	xSetForceError:BOOL;
	diSetForceErrorNr:DINT;
	xUpdateErrorList: BOOL;
	xResetErrorWarning:BOOL;
	xHideObject:BOOL;	(* Dies muss aktiv gesetzt werden sobald ein Overlay Message Aktiv ist, ansonsten kann es Probleme geben mit der Annahme der Button *)
(* Sicherheitstüre Maschine und Lader *)
	xOpenSecurityDoorMachine:BOOL;				(* Aufforderung für das Öffnen der Sicherheitstüren *)
	xCloseSecurityDoorMachine:BOOL;				(* Aufforderung für das Schliessen der Sicherheitstüren *)
(* Sicherheitssignale *)
	iSetupMode:INT;								(* Einrichtbetriebswahlschalter
													1=Einrichtbetrieb A
													2=Einrichtbetrieb B
												*)
	xSetupOperateModeActive:BOOL;				(* FALSE=NormalBetrieb, TRUE=Einrichtbetrieb *)
	bStateSafetyCtrl:BYTE;							(*
													0=< Keine Meldung >
													1=< Maschine ist am aufstarten... >
													2=< FreigabeTaste drücken >
													3=< StartTaste drücken >
													4=< Maschinen- und LadeTüre schliessen >
													5=< MaschinenTüren schliessen >
													6=< LadeTüre schliessen >
													7=< Für Positionsfahrt StartTaste drücken   >
													8=< Für Drehbewegung StartTaste drücken  >
													9=< Funktion in Ausführung >
													10=< Funktion in Ausführung...MMI ist blockiert >
													11=< Achsenposition wird überprüft...MMI ist blockiert >
													12=< Servo für Z Achsen stehen nicht bereit >
													13=< Servo für T Achse steht nicht bereit >
													14=< Servo für X Achse steht nicht bereit >
													15=< Kühlmittelpumpe Überlastschutz aktiv >
													16=< Kühlmittelpumpe nicht angeschlossen >
													17=< AntriebSperrTaste deaktivieren >
													18=< Schlüsselschalter deaktivieren >
													19=< Not Aus Taster deaktivieren >
													20=< Zustimmschalter deaktivieren >
													21=< Zustimmschalter aktivieren oder Türen schliessen >
													22=< Zylinderbewegung EIN/AUS drücken >
													23=< Ventile EIN/AUS drücken >
													24=< Zustimmschalter anschliessen >
													25=< Automat in Ausführung >
													26=< Masch.Ref/Grundstellung in Ausführung >
													27=< WstkEntladen in Ausführung >
													28=< HandBetrieb in Ausführung >
													29=< MaschinenTüreOben schliessen >
													30=< MaschinenTüreUnten schliessen >
													31=< MaschinenTüreOben und LadeTüre schliessen >
													32=< MaschinenTüreUnten und LadeTüre schliessen >
												*)
	xHideSafetyCtrlMessage:BOOL;					(* Unterdrückung der Sicherheitsmeldungen "bStateSafetyCtrl" *)
	xNormalOperate_EnergyON:BOOL;
	xSetupOperateA_EnergyON:BOOL;
	xSetupOperateB_EnergyON:BOOL;
	xDeactivateLamp:BOOL;						(* Gilt für den Lampentest, damit der Ausgang nicht mit der Logik überschrieben wird *)
	xSecurityDoorOpen:BOOL;						(* Maschinentüren und/oder Ladetüre offen *)
	bMachineDoorUpState:BYTE;					(* Zustand der Maschinentüre oben 1=Geöffnet, 2=Geschlossen, 3=Fehlverhalten *)
	bMachineDoorChannel1State:BYTE;				(* Zustand des zweikanaligen Türschalter Türe Zu für Türe oben und unten Kanal 1 1=OFF, 2=ON *)
	bMachineDoorChannel2State:BYTE;				(* Zustand des zweikanaligen Türschalter Türe Zu für Türe oben und unten Kanal 2 1=OFF, 2=ON *)
	bMachineDoorUpOpenState:BYTE;				(* Zustand des Türschalter Türe Offen für Türe oben 1=OFF, 2=ON *)
	bMachineDoorInductiveSensorState:BYTE;		(* Zustand des induktiven Sensor für Türe oben 1=OFF, 2=ON *)
	bMachineDoorGuardControlState:BYTE;			(* Zustand der Tür oben Zuhaltung 1=OFF, 2=ON *)
	iMsgInfo_ColourState:INT;						(* 0=Grün, 1=Gelb-->Gelb gilt für Prozess beendet mit mindestens einem Loch NoGo *)
END_STRUCT
END_TYPE

(* Data type in VISUALISIERUNG *)
TYPE ST_EXCHG_SPINDLEBURNIN :
STRUCT
	rTimeActive:REAL;
	rTimeInactive:REAL;
	rTimeMaxActiveFunction:REAL;
	rSpeed_Axis_S:REAL;
	tTimeElapsed:TIME;
END_STRUCT
END_TYPE

(* Data type in VISUALISIERUNG *)
TYPE ST_EXCHG_STATION :
STRUCT
	xExist:BOOL;
	xActiv:BOOL;
	wState:WORD;
	iProfile:INT;
	diErrorNr:DINT;
	sProfileName:STRING(30);
	bAutomodeState:BYTE;
END_STRUCT
END_TYPE

(* Data type in VISUALISIERUNG *)
TYPE ST_EXCHG_STATION_COMMON :
STRUCT
(* State *)
	wState:DWORD;

	T_Param_Machine:ST_RETAIN_DATA_MACHINE;
	T_Param_StationWork:ST_RETAIN_DATA_STATIONWORK;	(* Gilt für MicroHead-  Station *)

	T_ToolCounter_St1:ST_EXCHG_PARAM_TOOLCOUNTER;			(* Braucht es wegen der Parameterliste im NormalBetrieb, da auf diese Parameter gleichzeitig zugegriffen werden muss *)
	T_WPCounter_St1:ST_EXCHG_PARAM_WPCOUNTER;				(* Braucht es wegen der Parameterliste im NormalBetrieb, da auf diese Parameter gleichzeitig zugegriffen werden muss *)

(* Page Quality *)
	T_Button_Quality_Backward:ST_EXCHG_TOUCHBUTTON;
	T_Button_Quality_Forward:ST_EXCHG_TOUCHBUTTON;
	T_Input_Quality_HoleNumber:ST_EXCHG_TOUCHINPUT;

(* Axis State *)
	bState_Axis_Z:BYTE;

(* Gilt für die Ersteinrichtung der Z Achse *)
	iZAxisFirstSetup_StepNr:INT;
	iZAxisFirstSetupStartButton_StepNr:INT;
	iZAxisFirstSetup_ShowObjectNr:INT;
	xInitial_FirstSetupZ:BOOL;		(* TRUE = Ersteinrichtung Z durchgeführt *)
	rZAxisFirstSetup_OffsetSpinToDeskTop:REAL;

	xBlockSelectAutoMode:BOOL;	(* Bei aktivem Prozess muss die Auswahl blockiert sein *)

	(* Disablen von Objekten, wenn es den SystemLevel braucht *)
	xSystemLevelActive:BOOL;

	bActiveStation_St1St2:BYTE;	(* 	0=Arbeitsstation St1St2 Automat nicht Aktiv
									1=Arbeitsstation St1St2 Automat Aktiv
									2=Arbeitsstation St1St2 Automat Fehler *)

(* Gilt für das Aufzeichnen der Rotationsdauer der Spindel *)
	tSpindelActiveRotationTime:TIME;
	iSpindelActiveRotationDay:INT;

	xOnlineValueModified_St1:BOOL;

	xToolSpindle_L_Connect:BOOL;

(* Auswahl der Zylinderkonfiguration *)
	bSelectCylinderConfig:BYTE;		(* 1=Auslenkzylinder, 2=Drehmomentzylinder *)
	bShowCylinderConfig:BYTE;		(* 1=Auslenkzylinder (SM), 2=Auslenkzylinder (L), 3=Drehmomentzylinder (SM), 4=Drehmomentzylinder (L) *)

(* Auswahl der Erst Einrichtung Z Achse *)
	bSelectZAxisProcedure:BYTE;		(* 1=Ersteinrichtung Relation Z-Achse zu oberes Führungsrohr, 2=Ersteinrichtung Z Achse *)
	xBlockSelectZAxisProcedure:BOOL;

(* Gilt für die Ersteinrichtung der Z Achse für die Relation zwischen Z Achse und oberes Führungsrohr *)
	iZAxisGuideTube_StepNr:INT;
	iZAxisGuideTubeStartButton_StepNr:INT;
	iZAxisGuideTube_ShowObjectNr:INT;

(* Bestimmung der Schwingungsqualität der Wippe der Drehmomentüberwachung *)
	rRockerQuality:REAL;
	rRockerQualityMin:REAL;
	rRockerQualityMax:REAL;
	rRockerAmplitude:REAL;
	rRockerAmplitudeMin:REAL;
	rRockerAmplitudeMax:REAL;
	rRockerPosition:REAL;
	diRockerCountHC:DINT;
	diRockerCountHCTime:DINT;

(* Konfiguration der Positionen *)
	iSelectConfigPosition:INT;
	xDisableConfigPosition:BOOL;


(* Regler *)
	rSpeedZ_V1:REAL;					(* IGS *)
	rSpeedZ_V3:REAL;					(* IGS *)
	rTorqueZ_S1:REAL;					(* IGS *)
	rTorqueZ_S4:REAL;					(* IGS *)

	iProgressBar_Torque:INT;				(* IGS *)
	iProgressBar_ZPos:INT;				(* IGS *)
	iProgressBar_ZVel:INT;				(* IGS *)

	xTorqueAfterHC_Min_Overlimit:BOOL;	(* IGS *)
	xTorqueAfterHC_Max_Overlimit: BOOL;	(* IGS *)

	rActual_Torque:REAL;			(* Aktuelles Drehmoment der Drehmomentfeder in mNm - Wechselkopf unabhängig *)	(* IGS *)
	rMaxTorque:REAL;					(* IGS *)

(* Zentrieren *)
	diCentringNumberHCinWindow:DINT;	(* Anzeigen des Zählerstandes wie oft HC in einem definierten Fenster schon eingetroffen ist *)
	xShowSelectCentringProcess:BOOL;	(* Auswahl des Zentrierprozess nur dann zeigen wenn effektiv der Zentrierprozess angewählt ist *)

	rPositionEndProcCalc:REAL;	(* Anzeige oder Eingabe für berechnete EndPosition *)
	xDisableChangeEndPos:BOOL;

	rCentringEndProcCalc:REAL;	(* Anzeige oder Eingabe für berechnete EndPosition *)
	xDisableCentringChangeEndPos:BOOL;

	bSelectShowIncValue:BYTE;	(* 0=Anzeigen der Bearb Ink Werte, 1=Anzeigen der Zentrier Ink Werte *)

	rController2_MinSpeed:REAL;

	rZPositionEndProc:REAL;

	xProcessCylindricalAreaActive:BOOL;

	xSControllerActive:BOOL;
	xOControllerActive:BOOL;
END_STRUCT
END_TYPE

(* Data type in VISUALISIERUNG *)
TYPE ST_EXCHG_TOUCHBUTTON :
STRUCT
	xActive:BOOL;
	xDisable:BOOL;
	xHide:BOOL;
	bState:BYTE;
END_STRUCT
END_TYPE

(* Data type in VISUALISIERUNG *)
TYPE ST_EXCHG_TOUCHINPUT :
STRUCT
	diInput1:DINT;
	diInput2:DINT;
	diInputMin:DINT;
	diInputMax:DINT;
	xDisable:BOOL;
	xChangeColour:BOOL;
END_STRUCT
END_TYPE

(* Data type in VISUALISIERUNG *)
TYPE ST_EXCHG_TOUCHSCREENBTPANEL :
STRUCT
	iNotMaskTextBt:INT;
	iActivBtLeft:INT;
	iStateBtLeft:INT;
	iActivBtRight:INT;
	iStateSetupLamp:INT;
	iStateButtonPage:INT;
	iSelectStationNumber:INT;
END_STRUCT
END_TYPE

(* Data type in VISUALISIERUNG *)
TYPE ST_EXCHG_TOUCHSCREENNAVPANEL :
STRUCT
	wState:WORD;
	wNotMasktext:WORD;
	wActivBt:WORD;
END_STRUCT
END_TYPE

(* Data type in VISUALISIERUNG *)
TYPE ST_EXCHG_VISU :
STRUCT
(* Message structure *)
	T_Message:ST_EXCHG_MESSAGE;
(* Error List Structure *)
	T_MsgErrorEnglish:ST_EXCHG_MESSAGE_LIST;
	T_MsgErrorDeutsch:ST_EXCHG_MESSAGE_LIST;
(* Level structure *)
	T_Level:ST_EXCHG_LEVEL;
(* Variable *)
	iQVisActivNewPage:INT:=0;
	iLoadingStartPage:INT:=1;
	iHeaderTitlePageNumber:INT;
	bActivStation:BYTE:=0;
	bActiveSetupMode:BYTE:=0;	(* 0=AutoMode, 1=SetupMode A, 2=SetupMode B, 3=SetupMode C *)
	bMachineState:BYTE;	(* 1=Ready, no movement, 2=busy function,process or actuator active, 4=Error *)
	xKey_Enter:BOOL;
	xKey_Escape:BOOL;
	xLoadingProcessDone:BOOL;
	sSWVersion:STRING(10):='V4620699';		(* V4620699.pro *)
	sQVisVersion:STRING(10):='V462069902';	(* V4620699_02.qpr-->wird per NovRAM definiert *)
	sHWVersion:STRING(10):='V462069902';		(* V4620699_02.tsm *)
	sIPAddress:STRING(23):='xxx.xxx.xxx.xxx.xxx.xxx';
	sSubNetMask:STRING(23):='xxx.xxx.xxx.xxx.xxx.xxx';
	sGatewayAddress:STRING(23):='xxx.xxx.xxx.xxx.xxx.xxx';
	sAmsNetID:STRING(23):='xxx.xxx.xxx.xxx.xxx.xxx';
	sHostName:STRING(23):='xxxxxxxxxxxxxxxxxxxxxxx';
	xDHCPActive:BOOL:=FALSE;
	xNoRemoteControlActive:BOOL;	(* TRUE = Kein Rechner an der CX2020 angeschlossen *)
	xActiveProcessState_St1St2:BOOL;	(* Ausgabe ob Prozesszustand Aktiv ist oder nicht *)
END_STRUCT
END_TYPE

(* Data type in VISUALISIERUNG *)
TYPE ST_PAGE :
STRUCT
	iIndexConfigPage:INT:=0;
END_STRUCT
END_TYPE

(* Data type in VISUALISIERUNG *)
TYPE ST_QVIS :
STRUCT
	T_PageIndex:ARRAY[0..999] OF ST_PAGE;
	T_ConfigPage:ARRAY[1..csiMaxPage] OF ST_CONFIGPAGE;
	T_CtrleVisu:ST_CTRLEVISU;
	T_PlcParam:ST_VISU_PLC_PARAM;
	T_CtrleAction:ST_CTRLEACTION;
	T_CtrleProcess:ST_CTRLEPROCESS;
END_STRUCT
END_TYPE

(* Data type in VISUALISIERUNG *)
TYPE ST_QVIS_EXCHG_PARAM :
STRUCT
	byOverride:BYTE;					(*Maschinengeschwindigkeit*)
	T_Visu:ST_EXCHG_VISU;
	T_TouchScreenBtPanel:ST_EXCHG_TOUCHSCREENBTPANEL;
	T_BtFunctionPanel:ST_EXCHG_BTFUNCTIONPANEL;
	T_BtParameterList:ST_EXCHG_BTPARAMETERLIST;
	T_TouchScreenNavPanel:ST_EXCHG_TOUCHSCREENNAVPANEL;
	T_Config:ST_EXCHG_CONFIG;
	T_TeachIn:ST_EXCHG_AXIS;
	T_Cylinder:ST_EXCHG_CYLINDER;
	T_Station1:ST_EXCHG_STATION;	(* BearbStation St1 *)
	T_StationCommon:ST_EXCHG_STATION_COMMON;
	T_FunctionCommon:ST_EXCHG_FUNCTION_COMMON;
	T_AnalogSensTorque:ST_EXCHG_ANALOGSENSOR;
	T_ProfileCommon:ST_EXCHG_PROFILE_COMMON;
	T_PartQuality:ST_EXCHG_PARTQUALITY;
	T_LampTest:ST_EXCHG_LAMPTEST;
	T_SpindleBurnIn:ST_EXCHG_SPINDLEBURNIN;
	T_SafetyCtrl:ST_EXCHG_SAFETY_CTRL;
	T_ParamBIOS:ST_EXCHG_PARAM_BIOS;
	xShutdownSystem:BOOL;
	xBIOSButton:BOOL;
	xBIOSButtonHide:BOOL;

	(* Spindelkopf Auswahl Beckhoff/Maxon *)
	xInputSelectAxisSuccesful:BOOL;								(* IGS *)
	xButtonSelect_S1:BOOL;			(* Maxon Spindel *)			(* IGS *)
	xButtonSelect_S2:BOOL;			(* Beckhoff Spindel L *)			(* IGS *)
	xButtonSelect_S3:BOOL;			(* Beckhoff Spindel M *)			(* IGS *)
	xButtonDisable:BOOL;											(* IGS *)
	xWriteSoEParameter:BOOL;									(* IGS *)
	bToolSpindleActive:BYTE;			(*	1 = Maxon Spindel
										2 = Beckhoff Spindel L
										3 = Beckhoff Spindel M *)
END_STRUCT
END_TYPE

(* Data type in VISUALISIERUNG *)
TYPE ST_QVISCTRLE :
STRUCT
	dwInCommand:DWORD;
	dwInCount:DWORD;
	dwInQVisCtrlAddress:DWORD;
	dwInParameterAddress:DWORD;
	dwOutCount:DWORD;
	diOutStatus:DINT;
END_STRUCT
END_TYPE

(* Data type in VISUALISIERUNG *)
TYPE ST_TEMP_ACTIVE_STATE :
STRUCT
	iActCyl_SetupB1_St1:INT;		(* Cyl 1, Cyl 2, Cyl 3 *)

	iActValve_SetupB1_St1:INT;		(* Valve 4, Valve 5 *)

	iActCylinderSetup_SetupB1:INT;

	iActAxis_SetupB1_St1:INT;		(* Z, S und O Achse *)

	iActiveProfile:INT;
	iPtrListProfile:INT;
END_STRUCT
END_TYPE

(* Data type in VISUALISIERUNG *)
TYPE ST_VISU_PLC_PARAM :
STRUCT
	dwSetNewPage:DWORD;
	dwActualPage:DWORD;
	dwPreviousPage:DWORD;
END_STRUCT
END_TYPE

(* Data type in VISUALISIERUNG *)
TYPE ST_VISUPAGENUMBER :
STRUCT
(* Start Page *)
	iStart_Page1:INT:=0;
(* BIOS Page *)
	iBIOS_Page1:INT:=1;
	iBIOS_Page2:INT:=2;
(* NormalOperating-->Task 1 *)
	iAutoMode_Process:INT:=10;
	iAutoMode_ProcessValue1:INT:=11;		(* IGS *)
	iAutoMode_ProcessValue2:INT:=12;		(* IGS *)
	iAutoMode_PartQuality:INT:=13;			(* alt 12 *)
(* NormalOperating-->Task 2 *)
	iAutoMode_Referencing:INT:=20;
(* NormalOperating-->Task3 *)
	iAutoMode_Profile:INT:=30;
(* NormalOperating-->Task 4 *)
	iAutoMode_ToolChange:INT:=40;
	iAutoMode_UserLevel:INT:=41;
	iAutoMode_Language:INT:=42;
(* NormalOperating-->Task 5 *)
	iAutoMode_WPCounter:INT:=50;
	iAutoMode_LampTest:INT:=51;
	iAutoMode_SafetyCheck:INT:=52;
	iAutoMode_SysInfo:INT:=53;
(* NormalOperating-->Task 6 *)
	iAutoMode_ErrorList:INT:=60;
(* NormalOperating-->Parameter *)
	iAutoMode_Parameter:INT:=70;
(* SetupOperate A-->Task 1 *)
	iHandMode_Process:INT:=110;
	iHandMode_WorkParameter:INT:=111;	(* IGS *)
	iHandMode_RegulatorPara:INT:=112;	(* IGS *)
	iHandMode_OnlineChange:INT:=113;		(* alt 111 *)
	iHandMode_ConfigPosition:INT:=114;		(* alt 112 *)
(* SetupOperate A-->Task 3 *)
	iHandMode_ProfileMngmt1:INT:=120;
(* SetupOperate A-->Task 5 *)
	iHandMode_Setup1:INT:=150;
(* SetupOperate A-->Task 6 *)
	iHandMode_ErrorList:INT:=160;
(* SetupOperate A-->Parameter *)
	iHandMode_Parameter:INT:=170;
(* SetupOperate B-->Task 1 *)
	iWorkStation_Axis1:INT:=210;
(* SetupOperate B-->Task 2 *)
	iWorkStation_Cylinder1:INT:=220;
(* SetupOperate B-->Task 3 *)
	iWorkStation_Valve1:INT:=230;
(* SetupOperate B-->Task 4 *)
	iWorkStation_Function1:INT:=240;
(* SetupOperate B-->Task 5 *)
	iWorkStation_Setup1:INT:=250;
	iWorkStation_Setup2:INT:=251;
	iWorkStation_Setup3:INT:=252;
	iWorkStation_Setup4:INT:=253;
	iWorkStation_Setup5:INT:=254;
(* SetupOperate B-->Task 6 *)
	iWorkStation_ErrorList:INT:=260;
(* SetupOperate B-->Parameter *)
	iWorkStation_Parameter:INT:=270;
(* WaitCom_Page1 *)
	iWaitCom_Page1:INT:=1001;
END_STRUCT
END_TYPE

(* POU PRG_STARTUP, ST *)
PROGRAM PRG_STARTUP
VAR
	xPLCWait: BOOL := TRUE;
	TONPLCWait: TON;
	FBInitErrorList:FB_InitErrorList;
	RisingEdgeExecute:R_TRIG;
	iStepFunction: INT;
	xInitVisu: BOOL;
	tTimeOutFunction: TIME;
	xLoading: BOOL;
	TONStartUp: TON;
	xEmergency: BOOL;
	xStartBooting: BOOL;
	xNoAirPressure: BOOL;
	xReadHardware: BOOL;
	xActiveErrorMsg: BOOL;
	iMsgNumber: INT;
	xActiveInfoMsg: BOOL;
	TimerFunction: TON;
	xNovRamParameterReaded: BOOL;
	xTmp: BOOL;
	TONWaitResetOutput: TON;
	RisingEdgeStartButton: R_TRIG;
	RisingEdgeQuitButton: R_TRIG;
	xDeleteErrorMessage: BOOL;
	TONWaitCircuitOn: TON;
	xMsgActiveDeactivatedSupply: BOOL;
	xStationErrorActive: BOOL;
	tTimeStartUp: TIME := T#40ms;
	xActiveBootingError: BOOL;
	xForceCloseMessage: BOOL;
	xActiveWarningMsg: BOOL;
	xSetOutputDisable: BOOL;
	iStepFunctionMsg: INT;
	xActiveInfoMsgIntern: BOOL;
	xActiveErrorMsgIntern: BOOL;
	xActiveWarningMsgIntern: BOOL;
	TONWaitMessage: TON;
	iStepFunctionON: INT;
	TONWaitSetSecStateON: TON;
	xSwitchOffStartUpFunction: BOOL;
	xMachineActivated: BOOL;
	iStepUPS: INT;
	xFallingEdgeEnergyOff:BOOL;
	xRisingEdgeEnergyOn:BOOL;
	TONWaitEndMessage: TON;
	RisingEdgePower_SetupA_St1: R_TRIG;
	FallingEdgePower_SetupA_St1: F_TRIG;
	RisingEdgePower_SetupB_St1: R_TRIG;
	FallingEdgePower_SetupB_St1: F_TRIG;
	FBSafetyLogic: FB_SAFETYLOGIC;
	ptrTCommonAxis : POINTER TO ST_AXIS;
	xInitPointer: BOOL;
	FBCheckMachineState: FB_CHECKMACHINESTATE;
	iStepCheckSafetyError: INT;
	xTwinSAFEError: BOOL;
	xCheckConfirm: BOOL;
	xTerminalError: BOOL;
	RisingEdgePower_NormalOperate_St1St2: R_TRIG;
	FallingEdgePower_NormalOperate_St1St2: F_TRIG;
	FBGetAdaptersInfo: FB_GetAdaptersInfo;
	ii: INT;
	xReadyToCheckSafety: BOOL;
	xFirstBooting: BOOL;
	fbNT_Shutdown: NT_Shutdown;
	FBBIOSPARAMETER: FB_BIOSPARAMETER;
	xNovRamError: BOOL;
	RisingEdgeOpenSecDoorMachine: R_TRIG;
	RisingEdgeCloseSecDoorMachine: R_TRIG;
	xOpenSecurityDoor: BOOL;
	xCloseSecurityDoor: BOOL;
	iStepOpenSecurityDoor: INT;
	TONWaitSecurityDoorLocked: TON;
	iStepCloseSecurityDoor: INT;
	xReadySetMessageDeactivate: BOOL;
	xReadySetMessageActivate: BOOL;
	TONWaitCheckAirPressure: TON;
	RisingEdgeUPS: R_TRIG;
	TONPrellen_ON: TON;
	TONPrellen_OFF: TON;
	xCabinDoorLocked: BOOL;
	xInitMachineLamp: BOOL;
	RisingEdgeFirstTime: R_TRIG;
	RisingEdgeSetupOperateMode: R_TRIG;
	xInit: BOOL;
	TPEnablingSwitch: TP;
	RisingEdgeCheckSwitchVibration: R_TRIG;
	TONWaitStopVibration: TON;
	wWCEPOS_State: WORD;
	wEtherCAT_2_State: WORD;
	xActivateEPOSPreOPMode: BOOL;
	FBGetHostName: FB_GetHostName;
	FBGetLocalAmsNetId: FB_GetLocalAmsNetId;
	sCopyString: STRING;
	iPoint: INT;
	sCopyStringIP: STRING;

	T_TwinSafeInWithoutHW:POINTER TO	ST_TWINSAFE_IN;
	T_TwinSafeOutWithoutHW:	POINTER TO ST_TWINSAFE_OUT;

	(* .StartUpFunction_Booting *)
	TONWaitMessage1: TON;		(* IGS *)
END_VAR
(****************************************************************************************************************************************************)
(**********      This Functionblock manage the booting of the machine and the security mangament of the machine during   ********)
(**********       the machine operating                           														    ************)
(****************************************************************************************************************************************************)
(* waiting 5 sec before starting *)
	IF xPLCWait THEN
		TONPLCWait(IN:=TRUE,PT:=T#5s);
		IF TONPLCWait.Q THEN
			TONPLCWait(IN:=FALSE);
			xPLCWait:=FALSE;
			T_StartUp.T_Ctrle.xExecute:=FALSE;
			T_StartUp.T_Ctrle.xDone:=FALSE;
			T_StartUp.T_Ctrle.xErr:=FALSE;
			T_StartUp.T_Ctrle.xReset:=FALSE;
			T_StartUp.T_State.xPLCReady:=FALSE;
			T_StartUp.T_Ctrle.iFunction:=0;
			T_StartUp.T_Ctrle.udiErrorID:=16#0;
			T_StartUp.T_State.xBlockChangeMovementVisu:=TRUE;
			T_StartUp.T_Ctrle.iMsgNumber:=0;
			(* activ function "Start PLC" *)
			T_StartUp.T_Ctrle.xExecute:=TRUE;
			T_StartUp.T_Ctrle.iFunction:=1;
			FBInitErrorList(T_ErrorList:= T_ErrorList);	(* Init Static Text for Error List *)
		END_IF;
		RETURN;
	END_IF;
	(* Start and Quit Button *)
	RisingEdgeStartButton(CLK:=IxStartButton);
	RisingEdgeQuitButton(CLK:=IxReleaseButton);
	(* IN<-->OUT --> für TwinSAFE Verbindung mit Standard IO zu Sicherheit IO *)
	TPEnablingSwitch(IN:=	T_TwinSafeIn.IxEnablingSwitchActiveCh1 AND T_TwinSafeIn.IxEnablingSwitchActiveCh2 AND
							(NOT(FBSafetyLogic.xMachineDoorClose)) AND T_StartUp.T_State.xCompleted, PT:=T#0.1s);
	QxTwinSafeReleaseButton:=(IxReleaseButton OR TPEnablingSwitch.Q) ;	(* Übergabe des IxReleaseButton an TwinSafe Logik *)
	CtrlPowerSupply;
	CtrlEmergency;
	CtrlSecurityDoor;
	CtrlSecurityState;
	CtrlBIOSParameter;
	CtrlMachineLamp;
	CtrlStartUpFunction;

	IF NOT(xEmergency) AND NOT(xNoAirPressure) AND NOT(xTerminalError) THEN
		StartUpFunction_Initialisation;
		StartUpFunction_ReadHW;
		StartUpFunction_Booting;
		StartUpFunction_Loading;
	END_IF;

	StartUpFunction_MessageActivate;
	StartUpFunction_Emergency;

(* Delete of the line error message *)
	IF xDeleteErrorMessage THEN
		xDeleteErrorMessage:=FALSE;
		T_ExchgParam.T_Visu.T_Message.sDynamicTextEnglish:='';
		T_ExchgParam.T_Visu.T_Message.sDynamicTextDeutsch:='';
		T_ExchgParam.T_Visu.T_Message.sDynamicTextFrancais:='';
		T_ExchgParam.T_Visu.T_Message.iState:=0;	(* Meldung löschen *)
	END_IF;

(* Set Output disabled *)
	IF xSetOutputDisable THEN
		T_TwinSafeCtrleOUT.xTwinSAFE_Run_1:=FALSE;	(* Stop TwinSafe Groupe *)
		TProcess.T_Ctrle.xEnable:=FALSE;
		QxCtrlLampStartButton:=FALSE;
		QxCtrlLampStopButton:=FALSE;
		QxCtrlLampReleaseButton:=FALSE;
		QxCtrlLampAxesCurrentOff:=FALSE;
		QxReadyToOperateMasterModul1:=FALSE;
		QxReadyToOperateMasterModul2:=FALSE;
		TStation_Work_St1.TControl.xEnable:=FALSE;
		T_ExchgParam.T_Visu.iLoadingStartPage:=1;
		(* confirm *)
		xSetOutputDisable:=FALSE;
	END_IF;

	IF NOT(gxBlockChangeMovementVisuActiveMessage) AND NOT(xEmergency) AND NOT(xNoAirPressure) AND NOT(xTerminalError) AND NOT(xActiveInfoMsg) AND NOT(xActiveInfoMsgIntern)
	AND NOT(xActiveErrorMsg) AND NOT(xActiveErrorMsgIntern) AND NOT(xActiveWarningMsg) AND NOT(xActiveWarningMsgIntern) AND NOT(xPLCWait) AND T_StartUp.T_State.xCompleted THEN
		T_StartUp.T_State.xBlockChangeMovementVisu:=FALSE;
	END_IF;

	IF gxHardwareOFF AND NOT(xInit) THEN
		xInit:=TRUE;

		T_TwinSafeInWithoutHW:=ADR(T_TwinSafeIn);
		T_TwinSafeOutWithoutHW:=ADR(T_TwinSafeOut);
		T_TwinSafeInWithoutHW^.IxAxesCurrentOffCh1:=TRUE;
		T_TwinSafeInWithoutHW^.IxAxesCurrentOffCh2:=TRUE;
		T_TwinSafeInWithoutHW^.IxCabinDoorClose:=TRUE;
		T_TwinSafeInWithoutHW^.IxCabinDoorCloseCh1:=TRUE;
		T_TwinSafeInWithoutHW^.IxCabinDoorCloseCh2:=TRUE;
		T_TwinSafeInWithoutHW^.IxEmergencyStopButtonCh1:=TRUE;
		T_TwinSafeInWithoutHW^.IxEmergencyStopButtonCh2:=TRUE;
		T_TwinSafeInWithoutHW^.IxReadyToOperateMasterModul1:=TRUE;
		T_TwinSafeInWithoutHW^.IxReadyToOperateMasterModul2:=TRUE;
		T_TwinSafeOutWithoutHW^.QxContactor24VCh1:=TRUE;
		T_TwinSafeOutWithoutHW^.QxContactor24VCh2:=TRUE;
		T_TwinSafeOutWithoutHW^.QxContactorMasterModul400VCh1:=TRUE;
		T_TwinSafeOutWithoutHW^.QxContactorMasterModul400VCh2:=TRUE;
		T_TwinSafeOutWithoutHW^.QxEnablingAxisSpindle_St1:=TRUE;
		T_TwinSafeOutWithoutHW^.QxEnablingSwitchLed:=TRUE;

		T_NovRam.T_Parameter.T_StationWork[gciStationSt1].T_AxisState.xReferencedZAxis:=TRUE;

	END_IF;
END_PROGRAM
ACTION CtrlBIOSParameter:
	IF T_StartUp.T_State.xPLCReady THEN
		xTmp:=	T_TwinSafeOut.QxContactorMasterModul400VCh1 AND T_TwinSafeOut.QxContactorMasterModul400VCh2 AND
				T_TwinSafeOut.QxContactor24VCh1;
		FBBIOSPARAMETER(	dwBIOSPasswordPage:= gT_PageNumber.iBIOS_Page1,
							dwBIOSParameterPage:= gT_PageNumber.iBIOS_Page2,
							xActiveCurrentAxes:=xTmp,
							xReadyToSwitchPasswordPage:=xStartBooting AND (iStepFunction <= 40) AND T_TwinSafeIn.IxEmergencyStopButtonCh1 AND T_TwinSafeIn.IxEmergencyStopButtonCh2,
							T_Visu:= T_VisuQVis,
							T_ExchgParam:=T_ExchgParam,
							T_HDD:= T_HDD,
							T_NovRam:= T_NovRam,
							T_CtrlePanel:= T_CtrlePanel);
	END_IF;
END_ACTION
ACTION CtrlEmergency:
(* check the emergency stop, the air pressure, Lightbus of the MasterAxis after booting the machine *)

	IF T_StartUp.T_State.xPLCReady AND NOT(gxHardwareOFF) THEN
	(* check emergency stop, only if it is not already in this state *)
		IF NOT(T_TwinSafeIn.IxEmergencyStopButtonCh1) OR NOT(T_TwinSafeIn.IxEmergencyStopButtonCh2) THEN
			RisingEdgeExecute(CLK:=FALSE);
			(* Set emergency function *)
			T_StartUp.T_Ctrle.xExecute:=TRUE;
			T_StartUp.T_Ctrle.iFunction:=4;
			xSwitchOffStartUpFunction:=TRUE;
		END_IF;

	(* check air pressure, only if it is not already in this state *)
		IF NOT(IxAirSupply) AND T_TwinSafeOut.QxContactor24VCh1 AND T_TwinSafeOut.QxContactor24VCh2 THEN
			TONWaitCheckAirPressure(IN:=T_TwinSafeOut.QxContactor24VCh1 AND T_TwinSafeOut.QxContactor24VCh2,PT:=T#2s);
			IF TONWaitCheckAirPressure.Q THEN
				TONWaitCheckAirPressure(IN:=FALSE);
				(* Set No Air pressure function *)
				T_StartUp.T_Ctrle.xExecute:=TRUE;
				T_StartUp.T_Ctrle.iFunction:=6;
				xSwitchOffStartUpFunction:=TRUE;
			END_IF;
		ELSE
			TONWaitCheckAirPressure(IN:=FALSE);
		END_IF;

		IF xActivateEPOSPreOPMode THEN
			wWCEPOS_State:=8;
			wEtherCAT_2_State:=0;
		ELSE
			wWCEPOS_State:=T_TerminalState.wWCEPOS_State;
			wEtherCAT_2_State:=T_TerminalState.wEtherCAT_2_State;
		END_IF;
	(* Beckhoff Klemmen oder Koppler Überprüfung oder Power Supply 24V *)
		IF NOT(gxHardwareOFF) THEN
			xTmp:=	(T_TerminalState.wEtherCAT_1_State <> 0) OR (wEtherCAT_2_State <> 0) OR (T_TerminalState.wWCMasterAxisModul1_State <> 8) OR (T_TerminalState.wWCMasterAxisModul2_State <> 8)
					OR (wWCEPOS_State <> 8) OR (T_TerminalState.wWCSMCValve <> 8) OR NOT(IxFuse24VDC_OK);
		ELSE
			xTmp:=	FALSE;
		END_IF;
		IF xTmp THEN
			(* Set Terminal Error *)
			T_StartUp.T_Ctrle.xExecute:=TRUE;
			T_StartUp.T_Ctrle.iFunction:=3;
			xSwitchOffStartUpFunction:=TRUE;
		END_IF;

	(* Disable the active StartUp Function *)
		IF xSwitchOffStartUpFunction THEN
			xSwitchOffStartUpFunction:=FALSE;
			xInitVisu:=FALSE;
			xLoading:=FALSE;
			xStartBooting:=FALSE;
			xActiveErrorMsg:=FALSE;
			xActiveInfoMsg:=FALSE;
			xActiveWarningMsg:=FALSE;
			xNoAirPressure:=FALSE;
			xReadHardware:=FALSE;
			xTerminalError:=FALSE;
			T_StartUp.T_State.xCompleted:=FALSE;
		END_IF;
	END_IF;
END_ACTION
ACTION CtrlMachineLamp:
IF NOT(xInitMachineLamp) THEN
	xInitMachineLamp:=TRUE;
	TMachineLamp.T_CtrleCyl.xFBActiv:=TRUE;
	TMachineLamp.T_Config.xActivState:=TRUE;
	TMachineLamp.T_CtrleCyl.xReset:=TRUE;
END_IF;
RisingEdgeFirstTime(CLK:=T_StartUp.T_State.xPLCReady);
IF RisingEdgeFirstTime.Q OR RisingEdgeSetupOperateMode.Q THEN
	(* Einschalten der Einrichtlampe, nachdem die Maschine eingeschaltet wurde *)
	TMachineLamp.T_CtrleCyl.iFunction:=2;
	TMachineLamp.T_CtrleCyl.xExecute:=TRUE;
END_IF;
IF NOT(T_StartUp.T_State.xCompleted) AND T_StartUp.T_State.xPLCReady THEN
	(* Sollte z.B. wegen dem Not Aus die StartSeite wieder erreicht werden, dann muss die Lampe falls sie ausgeschaltet ist wieder eingeschaltet werden *)
	IF NOT(TMachineLamp.T_CtrleCyl.T_Standard.xActivOn) AND NOT(TMachineLamp.T_CtrleCyl.xExecute) AND TMachineLamp.T_CtrleCyl.xDone THEN
		TMachineLamp.T_CtrleCyl.iFunction:=2;
		TMachineLamp.T_CtrleCyl.xExecute:=TRUE;
	END_IF;
END_IF;
END_ACTION
ACTION CtrlPowerSupply:
RisingEdgeUPS(CLK:=TStatusUPS.ePowerStatus = PowerOnBattery);
IF RisingEdgeUPS.Q OR T_ExchgParam.xShutdownSystem THEN
	CASE iStepUPS OF
	1:	T_CtrleUPS.xBlockSystem_PowerFail:=TRUE;	(* Schicht 5 wird gesperrt *)
		T_TwinSafeCtrleOUT.xTwinSAFE_Run_1:=FALSE;	(* Stop TwinSafe Groupe 1 *)
		TProcess.T_Ctrle.xEnable:=FALSE;
		TStation_Work_St1.TControl.xEnable:=FALSE;
		xSwitchOffStartUpFunction:=FALSE;
		xInitVisu:=FALSE;
		xLoading:=FALSE;
		xStartBooting:=FALSE;
		xActiveErrorMsg:=FALSE;
		xActiveInfoMsg:=FALSE;
		xActiveWarningMsg:=FALSE;
		xNoAirPressure:=FALSE;
		xTerminalError:=FALSE;
		xReadHardware:=FALSE;
		T_StartUp.T_State.xCompleted:=FALSE;
		xActiveErrorMsgIntern:=TRUE;
		iStepFunctionMsg:=1;
		IF RisingEdgeUPS.Q THEN
			iMsgNumber:=51;		(* Stromausfall Detektiert! Daten werden im NovRAM gespeichert!! Steuerung ist blockiert! *)
		ELSIF T_ExchgParam.xShutdownSystem THEN
			iMsgNumber:=47;		(* System wird heruntergefahren! Daten werden im NovRAM gespeichert!! Steuerung ist blockiert! *)
		END_IF;
		IF xMachineActivated THEN
			iStepUPS:=iStepUPS + 1;
		ELSE
			fbNT_Shutdown(	NETID:= '127.0.0.1.1.1',
							DELAY:= 1,
							START:= FALSE,
							TMOUT:= T#10s);
			iStepUPS:=4;
		END_IF;
	(* NovRAM speichern *)
	2:	IF NOT(T_NovRAM.T_Ctrle.xExecute) AND (T_NovRAM.T_Ctrle.xDone OR T_NovRAM.T_Ctrle.xErr) THEN
			T_NovRAM.T_Ctrle.xExecute:=TRUE;
			T_NovRAM.T_Ctrle.iFunction:=2;
			iStepUPS:=iStepUPS + 1;
		END_IF;
	3:	IF NOT(T_NovRAM.T_Ctrle.xExecute) AND (T_NovRAM.T_Ctrle.xDone OR T_NovRAM.T_Ctrle.xErr) THEN
			iStepUPS:=iStepUPS + 1;
			fbNT_Shutdown(	NETID:= '127.0.0.1.1.1',
							DELAY:= 1,
							START:= FALSE,
							TMOUT:= T#10s);
		END_IF;
	4:	IF NOT(T_NovRAM.T_Ctrle.xExecute) AND (T_NovRAM.T_Ctrle.xDone OR T_NovRAM.T_Ctrle.xErr) THEN
			fbNT_Shutdown(	NETID:='127.0.0.1.1.1',
							DELAY:= 1,
							START:= TRUE,
							TMOUT:= T#10s);
			IF NOT(fbNT_Shutdown.BUSY) OR fbNT_Shutdown.ERR OR T_ExchgParam.xShutdownSystem THEN
				iStepUPS:=99;	(* CPU kann nun heruntergefahren werden *)
			END_IF;
		END_IF;
	END_CASE;
ELSE
	iStepUPS:=1;
END_IF;
END_ACTION
ACTION CtrlSecurityDoor:
RisingEdgeOpenSecDoorMachine(CLK:=T_ExchgParam.T_SafetyCtrl.xOpenSecurityDoorMachine);
RisingEdgeCloseSecDoorMachine(CLK:=T_ExchgParam.T_SafetyCtrl.xCloseSecurityDoorMachine);
IF RisingEdgeOpenSecDoorMachine.Q THEN
	xOpenSecurityDoor:=TRUE;
	xCloseSecurityDoor:=FALSE;
	T_ExchgParam.T_SafetyCtrl.xCloseSecurityDoorMachine:=FALSE;
END_IF;
IF RisingEdgeCloseSecDoorMachine.Q THEN
	xOpenSecurityDoor:=FALSE;
	xCloseSecurityDoor:=TRUE;
	T_ExchgParam.T_SafetyCtrl.xOpenSecurityDoorMachine:=FALSE;
END_IF;
TONPrellen_ON(IN:=IxCabinDoorLocked,PT:=T#50ms);
TONPrellen_OFF(IN:=NOT(IxCabinDoorLocked),PT:=T#50ms);
IF TONPrellen_ON.Q THEN
	xCabinDoorLocked:=TRUE;
END_IF;
IF TONPrellen_OFF.Q THEN
	xCabinDoorLocked:=FALSE;
END_IF;
IF xOpenSecurityDoor THEN
	CASE iStepOpenSecurityDoor OF
		1:	IF QxCabinDoorLock THEN
				xReadySetMessageDeactivate:=TRUE;
			END_IF;
			QxCabinDoorLock:=FALSE;
			TONWaitSecurityDoorLocked(IN:=FALSE);
			(* next step *)
			iStepOpenSecurityDoor:=iStepOpenSecurityDoor + 1;
		2:	TONWaitSecurityDoorLocked(IN:=TRUE,PT:=T#2000ms);
			IF TONWaitSecurityDoorLocked.Q OR (xCabinDoorLocked) THEN
				TONWaitSecurityDoorLocked(IN:=FALSE);
				(* next step *)
				iStepOpenSecurityDoor:=iStepOpenSecurityDoor + 1;
			END_IF;
		3:	xOpenSecurityDoor:=FALSE;
			T_ExchgParam.T_SafetyCtrl.xOpenSecurityDoorMachine:=FALSE;
			IF NOT(xCabinDoorLocked) THEN	(* IxCabinDoorUpLocked, Check if CabinDoor of the Machine is no more blocked *)
				T_ExchgParam.T_Visu.T_Message.iState:=287;	(* Kabinen-Türe Zuhaltung fehlerhaft beim öffnen ! *)
				xReadySetMessageDeactivate:=FALSE;
			END_IF;
			IF xReadySetMessageDeactivate THEN
				T_ExchgParam.T_Visu.T_Message.iState:=281;	(* Die Zuhaltung der Sicherheitstüren wurde deaktiviert! *)
			END_IF;
	END_CASE;
ELSE
	xReadySetMessageDeactivate:=FALSE;
	iStepOpenSecurityDoor:=1;
END_IF;
IF xCloseSecurityDoor THEN
	CASE iStepCloseSecurityDoor OF
		1:	IF NOT(QxCabinDoorLock) THEN
				xReadySetMessageActivate:=TRUE;
			END_IF;
			QxCabinDoorLock:=TRUE;
			TONWaitSecurityDoorLocked(IN:=FALSE);
			(* next step *)
			iStepCloseSecurityDoor:=iStepCloseSecurityDoor + 1;
		2:	TONWaitSecurityDoorLocked(IN:=TRUE,PT:=T#2000ms);
			IF TONWaitSecurityDoorLocked.Q OR NOT(xCabinDoorLocked) THEN
				TONWaitSecurityDoorLocked(IN:=FALSE);
				(* next step *)
				iStepCloseSecurityDoor:=iStepCloseSecurityDoor + 1;
			END_IF;
		3:	xCloseSecurityDoor:=FALSE;
			T_ExchgParam.T_SafetyCtrl.xCloseSecurityDoorMachine:=FALSE;
			IF xCabinDoorLocked THEN	(* IxCabinDoorUpLocked, Check if CabinDoor of the Machine is blocked *)
				T_ExchgParam.T_Visu.T_Message.iState:=286;	(* Kabinen-Türe Zuhaltung fehlerhaft beim schliessen ! *)
				xReadySetMessageActivate:=FALSE;
			END_IF;
			IF xReadySetMessageActivate THEN
				T_ExchgParam.T_Visu.T_Message.iState:=280;	(* Die Zuhaltung der Sicherheitstüren wurde aktiviert! *)
			END_IF;
	END_CASE;
ELSE
	xReadySetMessageActivate:=FALSE;
	iStepCloseSecurityDoor:=1;
END_IF;
END_ACTION
ACTION CtrlSecurityState:
	IF NOT(xInitPointer) THEN
		xInitPointer:=TRUE;
		ptrTCommonAxis:=ADR(TStation_Work_St1.THWWorkStation.TAxisZ);
	END_IF;
(* Function for Switch on the Security State *)
	IF T_StartUp.T_Ctrle.xSetSecurityStateON THEN
		CASE iStepFunctionON OF
		1:	QxCtrlLampStartButton:=FALSE;
			QxCtrlLampStopButton:=FALSE;
			QxCtrlLampReleaseButton:=FALSE;
			QxCtrlLampAxesCurrentOff:=FALSE;
			TONWaitSetSecStateON(IN:=FALSE);
			iStepFunctionON:=2;
		2:	TONWaitSetSecStateON(IN:=TRUE,PT:=T#500ms);
			IF TONWaitSetSecStateON.Q THEN
				TONWaitSetSecStateON(IN:=FALSE);
				T_TwinSafeCtrleOUT.xTwinSAFE_Run_1:=FALSE;	(* Stop TwinSafe Groupe 1 *)
				iStepFunctionON:=3;
			END_IF;
		3:	TONWaitSetSecStateON(IN:=TRUE,PT:=T#500ms);
			IF TONWaitSetSecStateON.Q THEN
				TONWaitSetSecStateON(IN:=FALSE);
				iStepFunctionON:=4;
			END_IF;
		4:	T_TwinSafeCtrleOUT.xTwinSAFE_Run_1:=TRUE;	(* Start TwinSafe Groupe 1 *)
			T_StartUp.T_Ctrle.xSetSecurityStateON:=FALSE;
			TONWaitSetSecStateON(IN:=FALSE);
			iStepFunctionON:=1;
		END_CASE;
	ELSE
		iStepFunctionON:=1;
		TONWaitSetSecStateON(IN:=FALSE);
	END_IF;

(* Zustandsüberwachung und Zuordnung der Sicherheitssignale *)
FBSafetyLogic(	T_TwinSafeIn:=T_TwinSafeIn,
				T_TwinSafeOut:=T_TwinSafeOut,
				xActiveBooting:=xLoading,
				xActiveBootingError:=xActiveBootingError,
				xVisuFunctionActive:=(NOT(T_VisuQVis.T_CtrleAction.xDone) OR T_VisuQVis.T_CtrleAction.xFunctionActive),
				dwActualPage:= T_VisuQVis.T_PlcParam.dwActualPage,
				xOverlayMessageAcitve:=(T_ExchgParam.T_SafetyCtrl.bStateMessageError<>0) OR (T_ExchgParam.T_SafetyCtrl.bStateMessageInfo<>0) OR (T_ExchgParam.T_SafetyCtrl.bStateMessageWarning<>0),
				iStateMessage:=T_ExchgParam.T_Visu.T_Message.iState,
				TCommonAxis:=ptrTCommonAxis^);

IF gT_SafetyStatus.xSetupOperateModeActive THEN
	CASE T_ExchgParam.T_TeachIn.iSetup_AxisSel OF
	1:	ptrTCommonAxis:=ADR(TStation_Work_St1.THWWorkStation.TAxisZ);
	2,3:	ptrTCommonAxis:=ADR(TStation_Work_St1.THWWorkStation.TAxisS);
	ELSE
		ptrTCommonAxis:=ADR(TStation_Work_St1.THWWorkStation.TAxisZ);
	END_CASE
END_IF;

IF (T_ExchgParam.T_SafetyCtrl.bStateSafetyCtrl = 99) OR T_ExchgParam.T_Visu.T_Message.xShowMessageInfo OR
    T_ExchgParam.T_Visu.T_Message.xShowMessageInput OR T_ExchgParam.T_Visu.T_Message.xShowMessageWarning OR
    (T_ExchgParam.T_Visu.T_Message.iState = 401) THEN
	T_ExchgParam.T_SafetyCtrl.xHideSafetyCtrlMessage:=TRUE;	(* Sicherheitsstatusmeldung auf der Visualisierung unterdrücken *)
ELSE
	T_ExchgParam.T_SafetyCtrl.xHideSafetyCtrlMessage:=FALSE;
END_IF;

T_ExchgParam.T_SafetyCtrl.bStateSafetyCtrl:=FBSafetyLogic.bStateSafetyCtrl;		(* Ausgabe direkt an der Visualisierung um den Operator Mitteilen zu können, was er unternehmen muss damit er Prozess,Funktion usw. auslösen kann *)

(* Kontrollampe für Freigabe QxCtrlLampReleaseButton der Energieversorgung *)
IF NOT(T_ExchgParam.T_SafetyCtrl.xDeactivateLamp) THEN	(* Wenn Lampen Test Aktiv ist, dann muss dies gesperrt werden *)
	QxCtrlLampReleaseButton:=	NOT(gT_SafetyStatus.xEnergyONNormalMode OR gT_SafetyStatus.xEnergyONSetupModeASt1 OR
								gT_SafetyStatus.xEnergyONSetupModeBSt1) AND
								FBSafetyLogic.xSafetyNotActive AND T_TwinSafeCtrleOUT.xTwinSAFE_Run_1 AND T_StartUp.T_State.xPLCReady AND
								(gT_SafetyStatus.xSecurityDoorClose);
END_IF;

(* Check Power switch on/off from the security circuit for control the Station *)
	RisingEdgePower_NormalOperate_St1St2(CLK:=gT_SafetyStatus.xEnergyONNormalMode);
	FallingEdgePower_NormalOperate_St1St2(CLK:=gT_SafetyStatus.xEnergyONNormalMode);
	RisingEdgePower_SetupA_St1(CLK:=	gT_SafetyStatus.xEnergyONSetupModeASt1);
	FallingEdgePower_SetupA_St1(CLK:=gT_SafetyStatus.xEnergyONSetupModeASt1);
	RisingEdgePower_SetupB_St1(CLK:=gT_SafetyStatus.xEnergyONSetupModeBSt1);
	FallingEdgePower_SetupB_St1(CLK:=gT_SafetyStatus.xEnergyONSetupModeBSt1);

	IF T_StartUp.T_State.xCompleted THEN
		xTmp:=	RisingEdgePower_NormalOperate_St1St2.Q OR FallingEdgePower_NormalOperate_St1St2.Q OR
				RisingEdgePower_SetupA_St1.Q OR FallingEdgePower_SetupA_St1.Q OR
				RisingEdgePower_SetupB_St1.Q OR FallingEdgePower_SetupB_St1.Q;
		IF xTmp THEN
			TStation_Work_St1.TControl.xSecurityCircuitOn:=			RisingEdgePower_NormalOperate_St1St2.Q OR RisingEdgePower_SetupA_St1.Q OR RisingEdgePower_SetupB_St1.Q;
			TStation_Work_St1.TControl.xSecurityCircuitOff:=			FallingEdgePower_NormalOperate_St1St2.Q OR FallingEdgePower_SetupA_St1.Q OR FallingEdgePower_SetupB_St1.Q;
		END_IF;
	(* Message Energy on/off *)
		xRisingEdgeEnergyOn:=	RisingEdgePower_NormalOperate_St1St2.Q OR
								RisingEdgePower_SetupA_St1.Q OR RisingEdgePower_SetupB_St1.Q;

		xFallingEdgeEnergyOff:=	FallingEdgePower_NormalOperate_St1St2.Q OR
								FallingEdgePower_SetupA_St1.Q OR FallingEdgePower_SetupB_St1.Q;

		IF T_StartUp.T_State.xCompleted AND xFallingEdgeEnergyOff THEN
			IF (T_ExchgParam.T_Visu.T_Message.iState = 0) OR (T_ExchgParam.T_Visu.T_Message.iState = 228) THEN
				T_ExchgParam.T_Visu.T_Message.iState:=229;	(* Warnung: Die Energieversorgung ist AUS ! *)
				TONWaitEndMessage(IN:=FALSE);
				T_ExchgParam.T_StationCommon.xBlockSelectAutoMode:=FALSE;
			END_IF;
		END_IF;
		IF T_StartUp.T_State.xCompleted AND xRisingEdgeEnergyOn THEN
			IF (T_ExchgParam.T_Visu.T_Message.iState = 0) OR (T_ExchgParam.T_Visu.T_Message.iState = 229) OR (T_ExchgParam.T_Visu.T_Message.iState = 279) THEN
				T_ExchgParam.T_Visu.T_Message.iState:=228;	(* Warnung: Die Energieversorgung ist EIN ! *)
				TONWaitEndMessage(IN:=FALSE);
			END_IF;
		END_IF;

	END_IF;

(* Überprüfe Maschinenstatus damit die entsprechende LED auf der Visu ausgegeben werden kann *)
FBCheckMachineState(	xSecurityKey:= gT_SafetyStatus.xSetupOperateModeActive,
						iSetupMode:= gT_SafetyStatus.iSetupMode,
						xNormalOperate_EnergyON:= gT_SafetyStatus.xEnergyONNormalMode,
						xSetupOperateA_EnergyON:= gT_SafetyStatus.xEnergyONSetupModeASt1,
						xSetupOperateB_EnergyON:= gT_SafetyStatus.xEnergyONSetupModeBSt1);
T_ExchgParam.T_SafetyCtrl.xNormalOperate_EnergyON:=	gT_SafetyStatus.xEnergyONNormalMode;
T_ExchgParam.T_SafetyCtrl.xSetupOperateA_EnergyON:=	gT_SafetyStatus.xEnergyONSetupModeASt1;
T_ExchgParam.T_SafetyCtrl.xSetupOperateB_EnergyON:=	gT_SafetyStatus.xEnergyONSetupModeBSt1;

(* Überwachung der Not Bremse für alle Achsen die am AX5206 angeschlossen sind beim ausschalten der Energieversorgung *)
	IF IxTwinSafeQuickStopMaster1_1 THEN	(* QuickStop Achsen von TwinSAFE *)
		QxEnableQuickStopMasterModul1:=TRUE;
	ELSE
		QxEnableQuickStopMasterModul1:=FALSE;	(* QxEnableQuickStopMasterModul1-->NotBremse aktivieren *)
	END_IF;
	IF IxTwinSafeQuickStopMaster2_1 OR IxTwinSafeQuickStopMaster2_2 THEN	(* QuickStop Achsen von TwinSAFE *)
		QxEnableQuickStopMasterModul2:=TRUE;
	ELSE
		QxEnableQuickStopMasterModul2:=FALSE;	(* QxEnableQuickStopMasterModul2-->NotBremse aktivieren *)
	END_IF;

(* Anzeigelampe für den EinrichtBetrieb *)
IF NOT(T_ExchgParam.T_SafetyCtrl.xDeactivateLamp) THEN	(* Wenn Lampen Test Aktiv ist, dann muss dies gesperrt werden *)
	IF gT_SafetyStatus.xSetupOperateModeActive AND T_StartUp.T_State.xCompleted THEN
		QxSetupModeLamp:=TRUE;
	ELSE
		QxSetupModeLamp:=FALSE;
	END_IF;
END_IF;

(* Anzeigelampe für AntriebSperrTaste *)
IF NOT(T_ExchgParam.T_SafetyCtrl.xDeactivateLamp) THEN	(* Wenn Lampen Test Aktiv ist, dann muss dies gesperrt werden *)
	IF T_TwinSafeIn.IxAxesCurrentOffCh1 AND T_TwinSafeIn.IxAxesCurrentOffCh2 THEN
		QxCtrlLampAxesCurrentOff:=FALSE;
	ELSE
		QxCtrlLampAxesCurrentOff:=TRUE;
	END_IF;
END_IF;

(* Überwachung ein TwinSAFE Fehler besteht *)
xTmp:=	(T_TwinSafeFBError.xMON_EmergencyButtonMachine OR				(* Diskrepanzfehler  Not Aus Taster Maschine *)
		T_TwinSafeFBError.xMON_Error_MachineDoor OR					(* Diskrepanzfehler Sicherheitstüre der Maschine *)
		T_TwinSafeFBError.xMON_KeySwitchProcObservation OR			(* Diskrepanzfehler Schlüsselschalter für Einrichtbetrieb Prozessbeobachtung Stellung I *)
		T_TwinSafeFBError.xMON_KeySwitchWorkStation OR				(* Diskrepanzfehler Schlüsselschalter für Einrichtbetrieb Bearbeitungsstation Stellung II *)
		T_TwinSafeFBError.xMON_EnablingSwitchActive OR					(* Diskrepanzfehler  Zustimmschalter *)
		T_TwinSafeFBError.xMON_AxesCurrentOff OR						(* Diskrepanzfehler Antriebsperrtaste *)
		T_TwinSafeFBError.xEDM_PowSup_MasterModul OR					(* Fehler im Rückführkreis der Leistungsschütze der  Z1 Achse (400V) *)
		T_TwinSafeFBError.xEDM_PowSup_24V OR							(* Fehler im Rückführkreis des Sicherheitsrelais für 24V Speisung *)
		((T_TwinSafeCtrleIN.xTwinSAFE_Group_OUT_Error_1 OR
		T_TwinSafeCtrleIN.xTwinSAFE_Group_FB_Error_1 OR
		T_TwinSafeCtrleIN.xTwinSAFE_Group_COM_Error_1) AND NOT(xStartBooting) AND NOT(xInitVisu) AND NOT(xReadHardware))) AND
		T_TwinSafeCtrleOUT.xTwinSAFE_Run_1 AND xReadyToCheckSafety;


IF (xTmp OR xTwinSAFEError) AND xNovRamParameterReaded THEN
	CASE iStepCheckSafetyError OF
	1:	xTwinSAFEError:=TRUE;
		T_VisuQVis.T_CtrleVisu.xReset:=TRUE;
		iStepCheckSafetyError:=iStepCheckSafetyError + 1;
		xSetOutputDisable:=TRUE;
	2:	IF NOT(T_VisuQVis.T_CtrleVisu.xReset) AND T_VisuQVis.T_CtrleVisu.xDone THEN
			IF T_TwinSafeFBError.xMON_EmergencyButtonMachine THEN
				iMsgNumber:=3;		(* Diskrepanzfehler zwischen den zweikanal. Schalter des Not Aus Taster der Maschine! Bitte Kontakt aufnehmen mit Microcut Ltd! *)
			ELSIF T_TwinSafeFBError.xMON_Error_MachineDoor THEN
				iMsgNumber:=4;		(* Diskrepanzfehler zwischen den zweikanal. Schalter der Sicherheitstüre der Maschine! Bitte Kontakt aufnehmen mit Microcut Ltd! *)
			ELSIF T_TwinSafeFBError.xMON_KeySwitchProcObservation THEN
				iMsgNumber:=5;		(* Diskrepanzfehler zwischen den zweikanal. Schalter des Schlüsselschalter Stellung I ! Bitte Kontakt aufnehmen mit Microcut Ltd! *)
			ELSIF T_TwinSafeFBError.xMON_KeySwitchWorkStation THEN
				iMsgNumber:=6;		(* Diskrepanzfehler zwischen den zweikanal. Schalter des Schlüsselschalter Stellung II ! Bitte Kontakt aufnehmen mit Microcut Ltd! *)
			ELSIF T_TwinSafeFBError.xMON_EnablingSwitchActive THEN
				iMsgNumber:=17;	(* Diskrepanzfehler zwischen den zweikanal. Schalter des Zustimmschalters! Bitte Kontakt aufnehmen mit Microcut Ltd! *)
			ELSIF T_TwinSafeFBError.xMON_AxesCurrentOff THEN
				iMsgNumber:=18;	(* Diskrepanzfehler zwischen den zweikanal. Schalter der AntriebSperrTaste! Bitte Kontakt aufnehmen mit Microcut Ltd! *)
			ELSIF T_TwinSafeFBError.xEDM_PowSup_MasterModul THEN
				iMsgNumber:=26;	(* Fehler im Rückführkreis des Schützes für Z1 Achse! Bitte Kontakt aufnehmen mit Microcut Ltd! *)
			ELSIF T_TwinSafeFBError.xEDM_PowSup_24V THEN
				iMsgNumber:=29;	(* Fehler im Rückführkreis des Sicherheitsrelais für Luftdruck und 24V Ausgänge Bitte Kontakt aufnehmen mit Microcut Ltd! *)
			ELSIF T_TwinSafeCtrleIN.xTwinSAFE_Group_OUT_Error_1 THEN
				iMsgNumber:=35;	(* TwinSAFE Sichere Ausgänge Fehlerhaft! Mindestens einen Sicheren Ausgang hat einen Fehler festgestellt! Bitte Kontakt aufnehmen mit Microcut Ltd! *)
			ELSIF T_TwinSafeCtrleIN.xTwinSAFE_Group_FB_Error_1 THEN
				iMsgNumber:=36;	(* TwinSAFE Funktionsbaustein Fehlerhaft! Mindestens ein Funktionsbaustein hat einen Fehler festgestellt! Bitte Kontakt aufnehmen mit Microcut Ltd! *)
			ELSIF T_TwinSafeCtrleIN.xTwinSAFE_Group_COM_Error_1 THEN
				iMsgNumber:=37;	(* TwinSAFE Sichere Verbindung Fehlerhaft! Mindestens eine Verbindung hat einen Fehler festgestellt! Bitte Kontakt aufnehmen mit Microcut Ltd! *)
			END_IF;
			(* Overlay Message Error *)
			xActiveErrorMsgIntern:=TRUE;
			iStepFunctionMsg:=1;
			iStepCheckSafetyError:=iStepCheckSafetyError + 1;
			TONWaitResetOutput(IN:=FALSE);
			xSwitchOffStartUpFunction:=FALSE;
			xLoading:=FALSE;
			xStartBooting:=FALSE;
			xActiveErrorMsg:=FALSE;
			xActiveInfoMsg:=FALSE;
			xActiveWarningMsg:=FALSE;
			xNoAirPressure:=FALSE;
			xTerminalError:=FALSE;
			T_StartUp.T_State.xCompleted:=FALSE;
			T_TwinSafeCtrleOUT.xTwinSAFE_Run_1:=TRUE;
		END_IF;
	3:	IF NOT(xActiveErrorMsgIntern) THEN
			iStepCheckSafetyError:=iStepCheckSafetyError + 1;
		END_IF;
	4:	TONWaitResetOutput(IN:=TRUE,PT:=T#0.2s);
		IF TONWaitResetOutput.Q THEN
			TONWaitResetOutput(IN:=FALSE);
			T_TwinSafeCtrleOUT.xTwinSAFE_Reset_1:=TRUE;
			iStepCheckSafetyError:=iStepCheckSafetyError + 1;
		END_IF;
	5:	TONWaitResetOutput(IN:=TRUE,PT:=T#0.2s);
		IF TONWaitResetOutput.Q THEN
			TONWaitResetOutput(IN:=FALSE);
			T_TwinSafeCtrleOUT.xTwinSAFE_Reset_1:=FALSE;
			iStepCheckSafetyError:=iStepCheckSafetyError + 1;
		END_IF;
	6:	IF NOT(xActiveErrorMsgIntern) THEN
			T_TwinSafeCtrleOUT.xTwinSAFE_Run_1:=FALSE;
			IF T_TwinSafeCtrleIN.xTwinSAFE_Group_OUT_Error_1 OR T_TwinSafeCtrleIN.xTwinSAFE_Group_FB_Error_1 OR T_TwinSafeCtrleIN.xTwinSAFE_Group_COM_Error_1 THEN
				iStepCheckSafetyError:=1;
				RETURN;
			END_IF;
			T_StartUp.T_Ctrle.xDone:=TRUE;
			T_StartUp.T_Ctrle.xErr:=FALSE;
			T_StartUp.T_Ctrle.udiErrorID:=0;
			(* Start Boot *)
			T_StartUp.T_Ctrle.xExecute:=TRUE;
			T_StartUp.T_Ctrle.iFunction:=5;
			xTwinSAFEError:=FALSE;
			iStepCheckSafetyError:=1;
		END_IF;
	END_CASE;
ELSE
	iStepCheckSafetyError:=1;
END_IF;

(* Vibrationssteuerung des Zustimmschalter *)
RisingEdgeCheckSwitchVibration(CLK:=T_TwinSafeOut.QxEnablingSwitchLed);
IF RisingEdgeCheckSwitchVibration.Q THEN
	QxEnablingSwitchVibration:=TRUE;
END_IF;
TONWaitStopVibration(IN:=QxEnablingSwitchVibration,PT:=T#0.5s);
IF TONWaitStopVibration.Q THEN
	QxEnablingSwitchVibration:=FALSE;
END_IF;
END_ACTION
ACTION CtrlStartUpFunction:
(****************************************************************************************************************************************************)
(***********                                               start of the management for calling of the start up function                                                   ************)
(****************************************************************************************************************************************************)
(* execute *)
	RisingEdgeExecute(CLK:=T_StartUp.T_Ctrle.xExecute);
	T_StartUp.T_Ctrle.xExecute:=FALSE;
	IF RisingEdgeExecute.Q THEN
		T_StartUp.T_Ctrle.xExecute:=FALSE;
		CASE T_StartUp.T_Ctrle.iFunction OF
		(* Start PLC *)
		1:	xInitVisu:=TRUE;
			tTimeOutFunction:=T#2s;
		(* Start loading *)
		2:	xLoading:=TRUE;
			T_ExchgParam.T_Visu.iLoadingStartPage:=1;
			tTimeOutFunction:=T#60s;
			TONStartUp(IN:=FALSE);
		(* Terminal Error *)
		3:	xTerminalError:=TRUE;
			tTimeOutFunction:=T#0s;	(* No Time out *)
			T_StartUp.T_State.xPLCReady:=FALSE;
		(* Emergency *)
		4:	xEmergency:=TRUE;
			tTimeOutFunction:=T#0s;	(* No Time out *)
			T_StartUp.T_State.xPLCReady:=FALSE;
		(* Start Booting *)
		5:	xStartBooting:=TRUE;
			tTimeOutFunction:=T#0s;	(* No Time out *)
		(* No Air pressure *)
		6:	xNoAirPressure:=TRUE;
			tTimeOutFunction:=T#0s;	(* No Time out *)
			T_StartUp.T_State.xPLCReady:=FALSE;
		(* Read NovRAM Parameter *)
		8:	xReadHardware:=TRUE;
			tTimeOutFunction:=T#5s;
		(* Activate Error Message Overlay *)
		10:	xActiveErrorMsg:=TRUE;
			iMsgNumber:=T_StartUp.T_Ctrle.iMsgNumber;
			tTimeOutFunction:=T#0s;	(* No Time out *)
			T_StartUp.T_State.xBlockChangeMovementVisu:=TRUE;	(* Lock the navigation of the visu *)
		(* Acitvate Info Message Overlay *)
		11:	xActiveInfoMsg:=TRUE;
			iMsgNumber:=T_StartUp.T_Ctrle.iMsgNumber;
			tTimeOutFunction:=T#0s;	(* No Time out *)
			T_StartUp.T_State.xBlockChangeMovementVisu:=TRUE;	(* Lock the navigation of the visu *)
		(* Activate Warning Message Overlay *)
		12:	xActiveWarningMsg:=TRUE;
			iMsgNumber:=T_StartUp.T_Ctrle.iMsgNumber;
			tTimeOutFunction:=T#0s;	(* No Time out *)
			T_StartUp.T_State.xBlockChangeMovementVisu:=TRUE;	(* Lock the navigation of the visu *)
		ELSE
		(* function not implemented *)
			T_StartUp.T_Ctrle.xDone:=FALSE;
			T_StartUp.T_Ctrle.xErr:=TRUE;
			T_StartUp.T_Ctrle.udiErrorID:=16#F000;
			(* Exit FB *)
			RETURN;
		END_CASE
		(* Init. variable *)
		iStepFunction:=1;
		iStepFunctionMsg:=1;
		T_StartUp.T_Ctrle.xDone:=FALSE;
		T_StartUp.T_Ctrle.xErr:=FALSE;
		T_StartUp.T_Ctrle.udiErrorID:=0;
		TimerFunction(IN:=FALSE);
		xCheckConfirm:=FALSE;
	(* Exit FB *)
		RETURN;
	END_IF
(****************************************************************************************************************************************************)
(***********                                               end of the management for calling of the start up function                                                   ************)
(****************************************************************************************************************************************************)
(* Time out function *)
	IF tTimeOutFunction <> T#0s THEN TimerFunction(IN:=TRUE,PT:=tTimeOutFunction); ELSE TimerFunction(IN:=FALSE); END_IF
	IF TimerFunction.Q AND NOT T_StartUp.T_Ctrle.xDone AND NOT T_StartUp.T_Ctrle.xErr THEN
	(* Error, timeout action activ *)
		T_StartUp.T_Ctrle.xErr:=TRUE;
		(* Display error message *)
		IF xInitVisu THEN
			iMsgNumber:=64;		(* TIMEOUT! Beim Aufstarten des Moduls konnte die Visualisierung nicht Initialisiert werden! Bitte Kontakt aufnehmen mit Microcut Ltd! *)
		ELSIF xReadHardware AND NOT(xNovRamError) THEN
			iMsgNumber:=65;		(* TIMEOUT! Beim Aufstarten des Moduls konnte die Hardware nicht Initialisiert werden! Bitte Kontakt aufnehmen mit Microcut Ltd! *)
		ELSIF xReadHardware AND xNovRamError THEN
			xNovRamError:=FALSE;
			iMsgNumber:=75;		(* TIMEOUT! Falsche Konfiguration des NovRAM Speicher! Hauptschalter  Aus! Bitte Kontakt aufnehmen mit Microcut Ltd! *)
		ELSIF xLoading THEN
			iMsgNumber:=66;		(* TIMEOUT! Beim Aufstarten des Moduls konnten die Stationen nicht Initialisiert werden! Bitte Kontakt aufnehmen mit Microcut Ltd! *)
		END_IF;
		xActiveErrorMsgIntern:=TRUE;
		iStepFunctionMsg:=1;
		iStepFunction:=1;
		(* Init. variable *)
		xInitVisu:=FALSE;
		xLoading:=FALSE;
		xReadHardware:=FALSE;
		(* Set output disable *)
		xSetOutputDisable:=TRUE;
		xCheckConfirm:=TRUE;
	END_IF
	IF xCheckConfirm AND NOT(xActiveErrorMsgIntern) THEN
		IF (iMsgNumber = 64) THEN
			(* Start InitVisu *)
			T_StartUp.T_Ctrle.xExecute:=TRUE;
			T_StartUp.T_Ctrle.iFunction:=1;
		ELSIF (iMsgNumber = 65) THEN
			(* Start ReadHardware *)
			T_StartUp.T_Ctrle.xExecute:=TRUE;
			T_StartUp.T_Ctrle.iFunction:=8;
		ELSIF (iMsgNumber = 66) THEN
			(* Start Booting *)
			T_StartUp.T_Ctrle.xExecute:=TRUE;
			T_StartUp.T_Ctrle.iFunction:=5;
		ELSIF (iMsgNumber = 75) THEN
			(* Start ReadHardware *)
			T_StartUp.T_Ctrle.xExecute:=TRUE;
			T_StartUp.T_Ctrle.iFunction:=8;
		END_IF;
	END_IF;
END_ACTION
ACTION StartUpFunction_Booting:
(* Function Start Booting *)
	IF xStartBooting THEN
		T_ExchgParam.T_Visu.iLoadingStartPage:=1;
		T_ExchgParam.xBIOSButtonHide:=FALSE;
		CASE iStepFunction OF
		1:	xDeleteErrorMessage:=TRUE;
			T_TwinSafeCtrleOUT.xTwinSAFE_Run_1:=FALSE;	(* Stop TwinSafe Groupe *)
			T_StartUp.T_State.xPLCReady:=FALSE;
			T_StartUp.T_State.xCompleted:=FALSE;
			QxCtrlLampStartButton:=FALSE;
			QxCtrlLampStopButton:=FALSE;
			QxReadyToOperateMasterModul1:=TRUE;
			QxReadyToOperateMasterModul2:=TRUE;
			T_HDD.T_Ctrle.xReset:=TRUE;
			IF T_VisuQVis.T_CtrleVisu.xQvis THEN	(* Visualisierung muss bereit stehen *)
				(* next step *)
				IF NOT(gxHardwareOFF) THEN
					(*iStepFunction:=10;*)
					iStepFunction:=iStepFunction+1;		(* IGS *)
				ELSE
					T_ExchgParam.xInputSelectAxisSuccesful:=TRUE;
					T_ExchgParam.bToolSpindleActive:=3;	(* Beckhoff Spindel M ausgewählt *)
					iStepFunction:=60;
					T_StartUp.T_State.xPLCReady:=TRUE;
				END_IF;
			END_IF;



		(* Auswahl treffen welche Spindel eingesetzt ist *)		(* IGS *)
		2:	(* next step *)
			IF NOT(T_ExchgParam.xInputSelectAxisSuccesful) THEN
				(* Der Operator muss zuerst eine Auswahl treffen ob Spindelkopf S1 oder Spindekopf S2 eingestetzt ist *)
				T_ExchgParam.xButtonSelect_S1:=FALSE;
				T_ExchgParam.xButtonSelect_S2:=FALSE;
				T_ExchgParam.xButtonSelect_S3:=FALSE;
				T_ExchgParam.xButtonDisable:=FALSE;
				iStepFunction:=iStepFunction+1;
			ELSE
				iStepFunction:=10;
			END_IF;
		3:	IF T_ExchgParam.xButtonSelect_S1 THEN	(* Maxon Spindel ausgewählt *)
				T_ExchgParam.xButtonSelect_S1:=FALSE;
				T_ExchgParam.xButtonDisable:=TRUE;
				T_ExchgParam.xWriteSoEParameter:=FALSE;
				T_ExchgParam.bToolSpindleActive:=1;
				TONWaitMessage1(IN:=FALSE);
				iStepFunction:=iStepFunction+1;
			END_IF;
			IF T_ExchgParam.xButtonSelect_S2 THEN	(* Beckhoff Spindel L ausgewählt *)
				T_ExchgParam.xButtonSelect_S2:=FALSE;
				T_ExchgParam.xButtonDisable:=TRUE;
				T_ExchgParam.xWriteSoEParameter:=TRUE;	(* -> LAYER2 -> FBHW_STATION_WORK.A01_AX5000_Parametrization -> Parameter schreiben durchführen *)
				T_ExchgParam.bToolSpindleActive:=2;
				TONWaitMessage1(IN:=FALSE);
				iStepFunction:=iStepFunction+1;
			END_IF;
			IF T_ExchgParam.xButtonSelect_S3 THEN	(* Beckhoff Spindel M ausgewählt *)
				T_ExchgParam.xButtonSelect_S3:=FALSE;
				T_ExchgParam.xButtonDisable:=TRUE;
				T_ExchgParam.xWriteSoEParameter:=TRUE;	(* -> LAYER2 -> FBHW_STATION_WORK.A01_AX5000_Parametrization -> Parameter schreiben durchführen *)
				T_ExchgParam.bToolSpindleActive:=3;
				TONWaitMessage1(IN:=FALSE);
				iStepFunction:=iStepFunction+1;
			END_IF;
		4:	CASE T_ExchgParam.bToolSpindleActive OF
			1:	(* Maxon Spindel *)
				TONWaitMessage1(IN:=TRUE,PT:=T#3s);
				T_ExchgParam.T_Visu.T_Message.iState:=79;	(* Info: Maxon Spindelkopf ausgewählt ! *)
				T_ExchgParam.T_Visu.T_Message.xShowMessageInfo:=TRUE;
				IF TONWaitMessage1.Q THEN
					TONWaitMessage1(IN:=FALSE);
					T_ExchgParam.xInputSelectAxisSuccesful:=TRUE;
					T_ExchgParam.T_Visu.T_Message.iState:=0;
					T_ExchgParam.T_Visu.T_Message.xShowMessageInfo:=FALSE;
					iStepFunction:=10;
				END_IF
			2:	(* Beckhoff Spindel L *)
				T_ExchgParam.T_Visu.T_Message.iState:=80;	(* Info: Beckhoff Spindelkopf L ausgewählt ! *)
				T_ExchgParam.T_Visu.T_Message.xShowMessageInfo:=TRUE;
				IF NOT(T_ExchgParam.xWriteSoEParameter) THEN
					T_ExchgParam.xInputSelectAxisSuccesful:=TRUE;
					T_ExchgParam.T_Visu.T_Message.iState:=0;
					T_ExchgParam.T_Visu.T_Message.xShowMessageInfo:=FALSE;
					iStepFunction:=10;
				END_IF
			3:	(* Beckhoff Spindel M *)
				T_ExchgParam.T_Visu.T_Message.iState:=81;	(* Info: Beckhoff Spindelkopf M ausgewählt ! *)
				T_ExchgParam.T_Visu.T_Message.xShowMessageInfo:=TRUE;
				IF NOT(T_ExchgParam.xWriteSoEParameter) THEN
					T_ExchgParam.xInputSelectAxisSuccesful:=TRUE;
					T_ExchgParam.T_Visu.T_Message.iState:=0;
					T_ExchgParam.T_Visu.T_Message.xShowMessageInfo:=FALSE;
					iStepFunction:=10;
				END_IF
			END_CASE;



		10:	T_TwinSafeCtrleOUT.xTwinSAFE_Run_1:=TRUE;	(* Start TwinSafe Groupe 1 *)
			TONWaitResetOutput(IN:=FALSE);
			(* next step *)
			iStepFunction:=11;
		11:	TONWaitResetOutput(IN:=TRUE,PT:=T#0.5s);
			IF TONWaitResetOutput.Q THEN
				IF T_TwinSafeCtrleIN.xTwinSAFE_Group_OUT_Error_1 OR T_TwinSafeCtrleIN.xTwinSAFE_Group_FB_Error_1 OR T_TwinSafeCtrleIN.xTwinSAFE_Group_COM_Error_1 THEN
					IF T_TwinSafeCtrleIN.xTwinSAFE_Group_OUT_Error_1 OR T_TwinSafeCtrleIN.xTwinSAFE_Group_FB_Error_1 OR T_TwinSafeCtrleIN.xTwinSAFE_Group_COM_Error_1 THEN
						T_TwinSafeCtrleOUT.xTwinSAFE_Reset_1:=TRUE;
					END_IF;
					TONWaitResetOutput(IN:=FALSE);
					iStepFunction:=12;
					RETURN;
				END_IF;
				TONWaitResetOutput(IN:=FALSE);
				iStepFunction:=14;
			END_IF;
		12:	TONWaitResetOutput(IN:=TRUE,PT:=T#0.2s);
			IF TONWaitResetOutput.Q THEN
				T_TwinSafeCtrleOUT.xTwinSAFE_Reset_1:=FALSE;
				TONWaitResetOutput(IN:=FALSE);
				iStepFunction:=13;
			END_IF;
		13:	TONWaitResetOutput(IN:=TRUE,PT:=T#0.2s);
			IF TONWaitResetOutput.Q THEN
				TONWaitResetOutput(IN:=FALSE);
				IF NOT(xFirstBooting) THEN
					iStepFunction:=10;
				ELSE
					iStepFunction:=14;
				END_IF;
			END_IF;
		14:	xReadyToCheckSafety:=TRUE;
			TStation_Work_St1.THWWorkStation.xActiveStation:=TRUE;
			TStation_Work_St1.TControl.xResetHardware:=TRUE;
			T_VisuQVis.T_CtrleVisu.xReset:=TRUE;
			T_VisuQVis.T_CtrleAction.xExecute:=FALSE;
			IF T_TwinSafeIn.IxReadyToOperateMasterModul1 AND T_TwinSafeIn.IxReadyToOperateMasterModul2 THEN
				iStepFunction:=17;
			ELSE
				iStepFunction:=15;	(* Mindestens eine Achse steht nicht Bereit-->Hardware wird zurückgesetzt *)
			END_IF;
		15:	IF NOT(TStation_Work_St1.TControl.xResetHardware) THEN
				iStepFunction:=16;
			END_IF;
		16:	IF T_TwinSafeIn.IxReadyToOperateMasterModul1 AND T_TwinSafeIn.IxReadyToOperateMasterModul2 THEN
				iStepFunction:=17;
			ELSE
				iStepFunction:=40;	(* Mindestens eine Achse steht immer noch nicht Bereit-->Fehlerausgabe *)
			END_IF;
		(* Überprüfe zuerst ob die USV bereit steht *)
		17:	IF T_CtrleUPS.xUPSReady THEN
				(* next step *)
				iStepFunction:=20;
			ELSE
				(* next step *)
				iStepFunction:=40;
			END_IF;
		20:	T_StartUp.T_State.xPLCReady:=TRUE;
			xFirstBooting:=TRUE;
			IF RisingEdgeQuitButton.Q OR gT_SafetyStatus.xEnergyONNormalMode THEN		(* Wait until the Operator press the external quit button *)
				xDeleteErrorMessage:=TRUE;	(* Reset the line message error *)
				TONWaitCircuitOn(IN:=FALSE);
				(* next step *)
				iStepFunction:=30;
			END_IF;
		30:	TONWaitCircuitOn(IN:=TRUE,PT:=T#1000ms);
			IF TONWaitCircuitOn.Q THEN
				TONWaitCircuitOn(IN:=FALSE);
				(* next step *)
				iStepFunction:=31;
			END_IF;
		31:	TStation_Work_St1.TControl.xResetHardware:=TRUE;
			iStepFunction:=iStepFunction + 1;
		32:	IF NOT(TStation_Work_St1.TControl.xResetHardware) THEN
				iStepFunction:=40;
			END_IF;
		40:	(* Overlay Message Error *)
			xActiveErrorMsgIntern:=TRUE;	(* Falls Kein Fehlverhalten festgestellt wird, dann wird es wieder zurückgesetzt *)
			iStepFunctionMsg:=1;
			iStepFunction:=50;
			iMsgNumber:=0;
			IF T_TwinSafeCtrleIN.xTwinSAFE_Group_OUT_Error_1 THEN
				iMsgNumber:=35;	(* TwinSAFE Sichere Ausgänge Fehlerhaft! Mindestens einen Sicheren Ausgang hat einen Fehler festgestellt! Bitte Kontakt aufnehmen mit Microcut Ltd!  *)
			ELSIF T_TwinSafeCtrleIN.xTwinSAFE_Group_FB_Error_1 THEN
				iMsgNumber:=36;	(* TwinSAFE Funktionsbaustein Fehlerhaft! Mindestens ein Funktionsbaustein hat einen Fehler festgestellt! Bitte Kontakt aufnehmen mit Microcut Ltd!  *)
			ELSIF T_TwinSafeCtrleIN.xTwinSAFE_Group_COM_Error_1 THEN
				iMsgNumber:=37;	(* TwinSAFE Sichere Verbindung Fehlerhaft! Mindestens eine Verbindung hat einen Fehler festgestellt! Bitte Kontakt aufnehmen mit Microcut Ltd! *)
			ELSIF NOT(T_CtrleUPS.xUPSReady) THEN
				iMsgNumber:=50;		(* Unterbrechungsfreie Stromversorgung USV steht nicht Bereit! Überprüfen Sie Bitte die USV und bestätigen Sie die Meldung *)
			ELSIF NOT(T_TwinSafeIn.IxReadyToOperateMasterModul1) THEN
				iMsgNumber:=39;		(* Achsen des MasterModul 1 stehen nicht Bereit! Überprüfen Sie Bitte den Servo des MasterModul 1 und bestätigen Sie die Meldung *)
			ELSIF NOT(T_TwinSafeIn.IxReadyToOperateMasterModul2) THEN
				iMsgNumber:=40;		(* Achsen des MasterModul 2 stehen nicht Bereit! Überprüfen Sie Bitte den Servo des MasterModul 2 und bestätigen Sie die Meldung *)
			ELSIF T_TwinSafeIn.IxKeySwitchProcObservationCh1 OR T_TwinSafeIn.IxKeySwitchProcObservationCh2 OR T_TwinSafeIn.IxKeySwitchWorkStationCh1 OR T_TwinSafeIn.IxKeySwitchWorkStationCh2 THEN
				iMsgNumber:=53;		(* Um die Maschine zu starten schalten Sie den Schlüsselschalter aus, bestätigen Sie die Meldung und drücken Sie erneut die StartTaste *)
			ELSIF NOT(T_TwinSafeIn.IxCabinDoorCloseCh1 AND T_TwinSafeIn.IxCabinDoorCloseCh2 AND NOT(T_TwinSafeIn.IxCabinDoorOpen) AND
			    T_TwinSafeIn.IxCabinDoorClose) THEN
				iMsgNumber:=54;		(* Um die Maschine zu starten schliessen Sie die MaschinenTüre, bestätigen Sie die Meldung und drücken Sie erneut die StartTaste *)
			ELSIF NOT(T_TwinSafeIn.IxAxesCurrentOffCh1) AND NOT(T_TwinSafeIn.IxAxesCurrentOffCh2) THEN
				iMsgNumber:=44;		(* Um die Maschine zu starten lösen Sie die AntriebSperrTaste, bestätigen Sie die Meldung und drücken Sie erneut die StartTaste *)
			ELSIF (NOT(T_TwinSafeOut.QxContactorMasterModul400VCh1) OR NOT(T_TwinSafeOut.QxContactorMasterModul400VCh2)) AND NOT(xMsgActiveDeactivatedSupply) AND NOT(xStationErrorActive) THEN
				iMsgNumber:=67;		(* Die Leistungsschütze der AX5106 Servos funktionieren nicht Einwandfrei! Bestätigen Sie die Meldung und versuchen Sie es erneut Kontrollieren Sie die Einrichtung *)
			ELSIF (NOT(T_TwinSafeOut.QxContactor24VCh1) OR NOT(T_TwinSafeOut.QxContactor24VCh2)) AND NOT(xMsgActiveDeactivatedSupply) AND NOT(xStationErrorActive) THEN
				iMsgNumber:=68;		(* Die Leistungsschütze der Luftversorgung und 24V funktionieren nicht Einwandfrei! Bestätigen Sie die Meldung und versuchen Sie es erneut Kontrollieren Sie die Einrichtung *)
			ELSIF (xMsgActiveDeactivatedSupply AND NOT(xStationErrorActive)) THEN
				iMsgNumber:=56;		(* Die Energieversorgung wurde ausgeschaltet! Bestätigen Sie die Meldung und versuchen Sie es erneut!  *)
			ELSIF xStationErrorActive THEN
				iMsgNumber:=49;		(* Während des Aufstarten der Maschine ist ein Fehler/Error aufgetreten! Bestätigen Sie die Meldung und Überprüfen Sie den entsprechenden Fehler/Error *)
			ELSE
				T_TwinSafeCtrleOUT.xTwinSAFE_Run_1:=TRUE;	(* Kein Fehlverhalten festgestellt, daher wird es wieder gesetzt *)
				xActiveErrorMsgIntern:=FALSE;						(* Kein Fehlverhalten festgestellt, daher wird es wieder zurückgesetzt *)
				TONWaitCircuitOn(IN:=FALSE);
				(* next step *)
				iStepFunction:=60;
			END_IF;
			IF (iMsgNumber <> 0) THEN
				T_TwinSafeCtrleOUT.xTwinSAFE_Run_1:=FALSE;	(* Stop TwinSafe Groupe-->Falls Kein Fehlverhalten festgestellt wird, dann wird es wieder gesetzt *)
			END_IF;
			xMsgActiveDeactivatedSupply:=xStationErrorActive:=FALSE;
			T_HDD.T_Ctrle.xReset:=TRUE;
		50:	IF NOT(xActiveErrorMsgIntern) THEN
				TONWaitCircuitOn(IN:=FALSE);
				IF QxCabinDoorLock THEN
					T_ExchgParam.T_SafetyCtrl.xOpenSecurityDoorMachine:=TRUE;
				ELSE
					T_ExchgParam.T_SafetyCtrl.xOpenSecurityDoorMachine:=FALSE;
				END_IF;
				(* next step *)
				iStepFunction:=51;
			END_IF;
		51:	IF NOT(T_ExchgParam.T_SafetyCtrl.xOpenSecurityDoorMachine) THEN
				(* next step *)
				iStepFunction:=1;
			END_IF;
		60:	QxCtrlLampStartButton:=TRUE;
			IF RisingEdgeStartButton.Q THEN		(* Wait until the Operator press the external start button *)
				QxCtrlLampStartButton:=FALSE;
				xDeleteErrorMessage:=TRUE;	(* Reset the line message error *)
				(* next step *)
				iStepFunction:=70;
			END_IF;
			IF (NOT(gT_SafetyStatus.xEnergyONNormalMode) OR NOT(gT_SafetyStatus.xSecuritySwitch)) AND NOT(gxHardwareOFF) THEN
				(* next step *)
				iStepFunction:=40;
				xMsgActiveDeactivatedSupply:=TRUE;
				QxCtrlLampStartButton:=FALSE;
				RETURN;
			END_IF;
		(* Aktivieren der Zuhaltung der Maschinen- Sicherheitstüre *)
		70:	T_ExchgParam.T_SafetyCtrl.xCloseSecurityDoorMachine:=TRUE;
			(* next step *)
			iStepFunction:=80;
		80:	IF NOT(T_ExchgParam.T_SafetyCtrl.xCloseSecurityDoorMachine) THEN
				iStepFunction:=90;
			END_IF;
		90:	(* Start Booting is ended, the machine has now the right state to boot the machine *)
			IF NOT(gT_SafetyStatus.xEnergyONNormalMode) AND NOT(gxHardwareOFF) THEN
				(* next step *)
				iStepFunction:=40;
				xMsgActiveDeactivatedSupply:=TRUE;
				RETURN;
			END_IF;
			xStartBooting:=FALSE;
			(* Start Loading *)
			T_StartUp.T_Ctrle.xExecute:=TRUE;
			T_StartUp.T_Ctrle.iFunction:=2;
		END_CASE;
	END_IF;
END_ACTION
ACTION StartUpFunction_Emergency:
(* Emergency or air supply *)
	IF (xEmergency OR xNoAirPressure OR xTerminalError) AND NOT(T_CtrleUPS.xBlockSystem_PowerFail) AND (TStatusUPS.ePowerStatus <> PowerOnBattery) THEN
		CASE iStepFunction OF
		1:	xSetOutputDisable:=TRUE;
			T_StartUp.T_State.xCompleted:=FALSE;
			T_NovRAM.T_Ctrle.xReset:=TRUE;
			T_StartUp.T_State.xBlockChangeMovementVisu:=TRUE;
			T_StartUp.T_Ctrle.xDeleteAllMessageOverlay:=TRUE;
			T_VisuQVis.T_CtrleAction.xDeleteVisuFunction:=TRUE;
			T_VisuQVis.T_CtrleVisu.xActive:=FALSE;
			T_StartUp.T_Ctrle.iMsgNumber:=0;
			TProcess.T_Ctrle.xError:=FALSE;
			iStepFunction:=iStepFunction + 1;
		2:	IF NOT(T_NovRAM.T_Ctrle.xReset) AND T_NovRAM.T_Ctrle.xDone THEN
				T_VisuQVis.T_CtrleVisu.xActive:=TRUE;
				iStepFunction:=iStepFunction + 1;
			END_IF;
		3:	IF T_VisuQVis.T_CtrleVisu.xActive AND T_VisuQVis.T_CtrleVisu.xDone THEN
				T_VisuQVis.T_CtrleVisu.xReset:=TRUE;
				iStepFunction:=iStepFunction + 1;
			END_IF;
		4:	IF NOT(T_VisuQVis.T_CtrleVisu.xReset) AND T_VisuQVis.T_CtrleVisu.xDone THEN
				T_VisuQVis.T_CtrleVisu.xReset:=TRUE;
				iStepFunction:=iStepFunction + 1;
			END_IF;
		(* waiting confirm *)
		5:	IF NOT(xSetOutputDisable) AND NOT(T_VisuQVis.T_CtrleVisu.xReset) THEN
				xActiveErrorMsgIntern:=TRUE;
				iStepFunctionMsg:=1;
				IF (T_TerminalState.wEtherCAT_1_State <> 0) THEN
					T_ExchgParam.T_SafetyCtrl.diSetForceErrorNr:=16#F100;	(* EtherCAT 1 Klemme Fehlerhaft *)
					iMsgNumber:=69;		(* Beckhoff Klemme oder Buskoppler Fehlerhaft! Herunterfahren der Steuerung, Modul ausschalten und schalten Sie dann das Modul wieder ein! *)
				ELSIF (wEtherCAT_2_State <> 0) THEN
					T_ExchgParam.T_SafetyCtrl.diSetForceErrorNr:=16#F101;	(* EtherCAT 2 Klemme Fehlerhaft *)
					iMsgNumber:=69;		(* Beckhoff Klemme oder Buskoppler Fehlerhaft! Herunterfahren der Steuerung, Modul ausschalten und schalten Sie dann das Modul wieder ein! *)
				ELSIF (wWCEPOS_State <> 8) THEN
					T_ExchgParam.T_SafetyCtrl.diSetForceErrorNr:=16#F102;	(* Maxon EPOS nicht im Operational Mode OP *)
					iMsgNumber:=69;		(* Beckhoff Klemme oder Buskoppler Fehlerhaft! Herunterfahren der Steuerung, Modul ausschalten und schalten Sie dann das Modul wieder ein! *)
				ELSIF (T_TerminalState.wWCSMCValve <> 8) THEN
					T_ExchgParam.T_SafetyCtrl.diSetForceErrorNr:=16#F103;	(* SMC Ventilinsel nicht im Operational Mode OP *)
					iMsgNumber:=69;		(* Beckhoff Klemme oder Buskoppler Fehlerhaft! Herunterfahren der Steuerung, Modul ausschalten und schalten Sie dann das Modul wieder ein! *)
				ELSIF (T_TerminalState.wWCMasterAxisModul1_State <> 8) THEN
					T_ExchgParam.T_SafetyCtrl.diSetForceErrorNr:=16#F104;	(* Achsen MasterModul 1 nicht im Operational Mode OP *)
					iMsgNumber:=69;		(* Beckhoff Klemme oder Buskoppler Fehlerhaft! Herunterfahren der Steuerung, Modul ausschalten und schalten Sie dann das Modul wieder ein! *)
				ELSIF (T_TerminalState.wWCMasterAxisModul2_State <> 8) THEN
					T_ExchgParam.T_SafetyCtrl.diSetForceErrorNr:=16#F105;	(* Achsen MasterModul 2 nicht im Operational Mode OP *)
					iMsgNumber:=69;		(* Beckhoff Klemme oder Buskoppler Fehlerhaft! Herunterfahren der Steuerung, Modul ausschalten und schalten Sie dann das Modul wieder ein! *)
				ELSIF NOT(IxFuse24VDC_OK) THEN
					T_ExchgParam.T_SafetyCtrl.diSetForceErrorNr:=16#F106;	(* Spannungsversorgung 24VDC fehlerhaft *)
					iMsgNumber:=59;		(* Spannungsversorgung 24VDC fehlerhaft! Herunterfahren der Steuerung, Maschine ausschalten und schalten Sie dann die Maschine wieder ein!  *)
				ELSIF (NOT(T_TwinSafeIn.IxEmergencyStopButtonCh1) OR NOT(T_TwinSafeIn.IxEmergencyStopButtonCh2)) THEN
					iMsgNumber:=1;		(* Not-Aus Taste Maschine ist betätigt! Lösen Sie die Not-Aus Taste und bestätigen Sie die Meldung *)
					T_ExchgParam.T_SafetyCtrl.diSetForceErrorNr:=1;	(* Not Aus Taste Maschine wurde gedrückt *)
				ELSIF xNoAirPressure THEN
					iMsgNumber:=2;		(* Keine Druckluft! Stellen Sie die Zufuhr sicher und bestätigen Sie die Meldung *)
					T_ExchgParam.T_SafetyCtrl.diSetForceErrorNr:=8;	(* Keine Druckluft *)
				END_IF;
				T_ExchgParam.T_SafetyCtrl.xSetForceError:=TRUE;
				iStepFunction:=iStepFunction + 1;
			END_IF
		6:	IF NOT(xActiveErrorMsgIntern) THEN
					wWCEPOS_State:=8;
					wEtherCAT_2_State:=0;
					IF (T_TerminalState.wEtherCAT_1_State <> 0) OR (wEtherCAT_2_State <> 0) OR (T_TerminalState.wWCMasterAxisModul1_State <> 8) OR (T_TerminalState.wWCMasterAxisModul2_State <> 8)
					OR (wWCEPOS_State <> 8) OR (T_TerminalState.wWCSMCValve <> 8) OR NOT(IxFuse24VDC_OK)THEN
					(* next step *)
					iStepFunction:=iStepFunction + 1;
					TONWaitMessage(IN:=FALSE);
				ELSIF NOT(T_TwinSafeIn.IxEmergencyStopButtonCh1) OR NOT(T_TwinSafeIn.IxEmergencyStopButtonCh2) THEN
					(* next step *)
					iStepFunction:=iStepFunction + 1;
					TONWaitMessage(IN:=FALSE);
				ELSE
					(* next step *)
					iStepFunction:=90;
				END_IF;
			END_IF;
		7:	TONWaitMessage(IN:=TRUE,PT:=T#1s);
			IF TONWaitMessage.Q THEN
				(* next step *)
				iStepFunction:=5;	(* NotAus immer noch gedrückt-->Wiederhole die Meldung *)
			END_IF;
		(* Check if the SecurityDoor is locked *)
		90:	IF NOT(IxCabinDoorLocked) THEN
				xActiveErrorMsgIntern:=TRUE;
				iStepFunctionMsg:=1;
				iMsgNumber:=48;		(* Die MaschinenTüre ist zugehalten Bestätigen Sie und die Zuhaltung Der MaschinenTüre wird deaktiviert *)
				(* next step *)
				iStepFunction:=iStepFunction + 1;
			ELSE
				(* next step *)
				iStepFunction:=99;
			END_IF;
		91:	IF NOT(xActiveErrorMsgIntern) THEN
				T_ExchgParam.T_SafetyCtrl.xOpenSecurityDoorMachine:=TRUE;
				(* next step *)
				iStepFunction:=iStepFunction + 1;
			END_IF;
		92:	IF NOT(T_ExchgParam.T_SafetyCtrl.xOpenSecurityDoorMachine) THEN
				iStepFunction:=99;
			END_IF;
		(* end function or time out *)
		99:	xActiveErrorMsg:=FALSE;
			xActiveInfoMsg:=FALSE;
			xActiveWarningMsg:=FALSE;
			T_StartUp.T_Ctrle.xDone:=TRUE;
			T_StartUp.T_Ctrle.xErr:=FALSE;
			T_StartUp.T_Ctrle.udiErrorID:=0;
			xEmergency:=FALSE;
			xNoAirPressure:=FALSE;
			xTerminalError:=FALSE;
			(* Start Boot *)
			T_StartUp.T_Ctrle.xExecute:=TRUE;
			T_StartUp.T_Ctrle.iFunction:=5;
		END_CASE
	END_IF;
END_ACTION
ACTION StartUpFunction_Initialisation:
(* Function Init PLC *)
	IF xInitVisu THEN
		CASE iStepFunction OF
		1:	T_VisuQVis.T_CtrleVisu.xActive:=TRUE;
			T_VisuQVis.T_CtrleVisu.xReset:=TRUE;
			(* next step *)
			iStepFunction:=10;
		(* Confirm Reset *)
		10:	IF T_VisuQVis.T_CtrleVisu.xDone THEN
				(* next step *)
				iStepFunction:=90;
			END_IF
		(* end function or time out *)
		90:	T_StartUp.T_Ctrle.xDone:=TRUE;
			T_StartUp.T_Ctrle.xErr:=FALSE;
			T_StartUp.T_Ctrle.udiErrorID:=0;
			xInitVisu:=FALSE;
			tTimeOutFunction:=T#0s;
			(* Start Read Hardware *)
			T_StartUp.T_Ctrle.xExecute:=TRUE;
			T_StartUp.T_Ctrle.iFunction:=8;
		END_CASE
	END_IF
END_ACTION
ACTION StartUpFunction_Loading:
(* Function start loading *)
	IF xLoading THEN
		(* Timer bargraph *)
		IF (iStepFunction < 999) THEN
			TONStartUp(IN:=TRUE,PT:=tTimeStartUp);
			IF TONStartUp.Q THEN
				TONStartUp(IN:=FALSE);
				IF (T_ExchgParam.T_Visu.iLoadingStartPage <=100) THEN
					T_ExchgParam.T_Visu.iLoadingStartPage:=T_ExchgParam.T_Visu.iLoadingStartPage +1; END_IF
			END_IF;
		END_IF;
		IF NOT(gT_SafetyStatus.xEnergyONNormalMode) AND (iStepFunction < 985) AND NOT(gxHardwareOFF) THEN
			T_ExchgParam.T_SafetyCtrl.diSetForceErrorNr:=9;		(* Spannungsversorgung wurde ausgeschaltet *)
			T_ExchgParam.T_SafetyCtrl.xSetForceError:=TRUE;
			iStepFunction:=999;
		END_IF;
		CASE iStepFunction OF
		(* Check *)
		1:	IF T_StartUp.T_State.xPLCReady THEN iStepFunction:=10; END_IF
			tTimeStartUp:=T#40ms;
		(* Init. Visu and Set Power *)
		10:	gxInitialStateActivated:=FALSE;
			xActiveBootingError:=FALSE;
			xDeleteErrorMessage:=TRUE;	(* Reset the line message error *)
			T_VisuQVis.T_PlcParam.dwSetNewPage:=16#0;
			T_VisuQVis.T_CtrleVisu.xReset:=TRUE;
			T_VisuQVis.T_CtrleVisu.xExecute:=TRUE;
			T_VisuQVis.T_CtrleVisu.iFunction:=1;
			(* next Step *)
			iStepFunction:=20;
		(* wait until the reset procedure is ready *)
		20:	IF NOT(T_VisuQVis.T_CtrleVisu.xReset) AND T_VisuQVis.T_CtrleVisu.xQvis THEN
				(* next Step *)
				IF NOT(gxHardwareOFF) THEN
					iStepFunction:=30;
				ELSE
					iStepFunction:=70;		(* IGS alt: 30; *)
				END_IF;
			END_IF;
		(* Adapter Informationen lesen *)
		30:	FBGetAdaptersInfo(	sNetID:= '',
								bExecute:=FALSE);
			iStepFunction:=40;
		40:	FBGetAdaptersInfo(	sNetID:= '',
								bExecute:= TRUE,
								tTimeout:= T#2s);
			IF NOT(FBGetAdaptersInfo.bBusy) THEN
				FOR ii:=0 TO UDINT_TO_INT(FBGetAdaptersInfo.nGet - 1) DO
					IF (FIND(FBGetAdaptersInfo.arrAdapters[ii].sDescription,'#2') <> 0) AND (FBGetAdaptersInfo.arrAdapters[ii].eType = MIB_IF_TYPE_ETHERNET) THEN
						T_ExchgParam.T_Visu.sIPAddress:=FBGetAdaptersInfo.arrAdapters[ii].sIpAddr;
						T_ExchgParam.T_Visu.sSubNetMask:=FBGetAdaptersInfo.arrAdapters[ii].sSubNet;
						T_ExchgParam.T_Visu.xDHCPActive:=FBGetAdaptersInfo.arrAdapters[ii].bDhcpEnabled;
						T_ExchgParam.T_Visu.sGatewayAddress:=FBGetAdaptersInfo.arrAdapters[ii].sDefGateway;
						EXIT;
					END_IF;
				END_FOR;
				FBGetHostName(	bExecute:=FALSE);
				iStepFunction:=41;
			END_IF;
		41:	FBGetHostName(	sNetID:= '',
								bExecute:= TRUE,
								tTimeout:= T#2s);
			IF NOT(FBGetHostName.bBusy) THEN
				T_ExchgParam.T_Visu.sHostName:=FBGetHostName.sHostName;
				FBGetLocalAmsNetId(	bExecute:=FALSE);
				iStepFunction:=42;
			END_IF;
		42:	FBGetLocalAmsNetId(	bExecute:= TRUE,
									tTimeout:= T#2s);
			IF NOT(FBGetLocalAmsNetId.bBusy) THEN
				T_ExchgParam.T_Visu.xNoRemoteControlActive:=FALSE;
				IF (FBGetLocalAmsNetId.AddrString <> '') AND NOT(FBGetLocalAmsNetId.bError) THEN
					T_ExchgParam.T_Visu.sAmsNetID:=FBGetLocalAmsNetId.AddrString;
					IF (FIND(STR1:=T_ExchgParam.T_Visu.sIPAddress, STR2:='0.0.0.0') <> 0) AND NOT(T_ExchgParam.T_Visu.xDHCPActive) THEN
						(* An der CX2020 ist am Netzwerkadapter kein Rechner angeschlossen und deshalb wird die konfigurierte IP Adresse nicht ausgegeben. Man geht davon aus dass die AmsNetID der IP Adresse entspricht und übergibt diesen ausser nicht den Byte 5 und 6 Wert nicht *)
						sCopyString:=FBGetLocalAmsNetId.AddrString;
						sCopyStringIP:='';
						FOR ii:=1 TO 4 DO
							iPoint:=FIND(STR1:=sCopyString, STR2:='.');
							sCopyStringIP:=CONCAT(sCopyStringIP,MID(STR:=sCopyString, LEN:=iPoint, POS:=1));
							sCopyString:=DELETE(STR:=sCopyString, LEN:=iPoint, POS:=1);
						END_FOR;
						sCopyStringIP:=DELETE(STR:=sCopyStringIP, LEN:=1, POS:=LEN(sCopyStringIP));	(* Den letzten Punkt muss gelöscht werden *)
						T_ExchgParam.T_Visu.sIPAddress:=sCopyStringIP;
						T_ExchgParam.T_Visu.sSubNetMask:='255.255.255.0';
						T_ExchgParam.T_Visu.xNoRemoteControlActive:=TRUE;	(* In diesem Fall werde die IP Adresse und Subnetmaske Orange dargestellt, dass es Möglich sein könnte dass es nicht dem eingestellten Wert entspricht *)
					END_IF;
				END_IF;
				iStepFunction:=50;
			END_IF;
		(* Überprüfe ob USB-Stick eingesteckt ist *)
		50:	T_Profile.T_Ctrle.iFunction:=3;		(* check if USB Stick exist *)
			T_Profile.T_Ctrle.xExecute:=TRUE;
			iStepFunction:=60;
		60:	IF NOT(T_Profile.T_Ctrle.xExecute) AND T_Profile.T_Ctrle.xDone THEN
				iStepFunction:=70;
			END_IF;
			IF NOT(T_Profile.T_Ctrle.xExecute) AND T_Profile.T_Ctrle.xErr THEN
				T_ExchgParam.T_SafetyCtrl.diSetForceErrorNr:=16#F305;	(* USB-Stick konnte nicht gefunden werden *)
				T_ExchgParam.T_SafetyCtrl.xSetForceError:=TRUE;
				T_Profile.T_Ctrle.xReset:=TRUE;
				iStepFunction:=999;
			END_IF;
		(* Lesen des Operator Passwortes *)
		70:	T_Password.T_Ctrle.xExecute:=TRUE;
			T_Password.T_Ctrle.iFunction:=1;
			iStepFunction:=80;
		80:	IF NOT(T_Password.T_Ctrle.xExecute) AND T_Password.T_Ctrle.xDone THEN
				T_ExchgParam.T_Visu.T_Level.diPwOperatorSaved:=T_Password.T_Ctrle.udiGetOperatorPassword;
				iStepFunction:=90;
			END_IF;
			IF NOT(T_Password.T_Ctrle.xExecute) AND T_Password.T_Ctrle.xErr THEN
				T_ExchgParam.T_Visu.T_Level.diPwOperatorSaved:=123456;	(* Bei Fehler Standardmässig Passwort 123456 definieren *)
				T_Password.T_Ctrle.xReset:=TRUE;
				iStepFunction:=90;
			END_IF;
		(* Überprüfe ob die Maschinenkonfiguration bezüglich der ausgewählten Stationen korrekt ist *)
		90:	iStepFunction:=100;
		100:	(* Aktivierung der Stationen *)
			TStation_Work_St1.TControl.xActiveStation:=TRUE;
			TStation_Work_St1.THWWorkStation.xActiveStation:=TRUE;
			TStation_Work_St1.THWWorkStation.TCtrlWork.iSpindelActiveRotationDay:=T_NovRAM.T_Parameter.T_StationWork[gciStationSt1].iSpindelActiveRotationDay;
			TStation_Work_St1.THWWorkStation.TCtrlWork.tSpindelActiveRotationTime:=T_NovRAM.T_Parameter.T_StationWork[gciStationSt1].tSpindelActiveRotationTime;
			TStation_Work_St1.THWWorkStation.TCtrlWork.iSpindel2ActiveRotationDay:=T_NovRAM.T_Parameter.T_StationWork[gciStationSt1].iSpindel2ActiveRotationDay;
			TStation_Work_St1.THWWorkStation.TCtrlWork.tSpindel2ActiveRotationTime:=T_NovRAM.T_Parameter.T_StationWork[gciStationSt1].tSpindel2ActiveRotationTime;
			TStation_Work_St1.THWWorkStation.TCtrlWork.iSpindel3ActiveRotationDay:=T_NovRAM.T_Parameter.T_StationWork[gciStationSt1].iSpindel3ActiveRotationDay;
			TStation_Work_St1.THWWorkStation.TCtrlWork.tSpindel3ActiveRotationTime:=T_NovRAM.T_Parameter.T_StationWork[gciStationSt1].tSpindel3ActiveRotationTime;
			TStation_Work_St1.TControl.xEnable:=TRUE;
			iStepFunction:=200;
		(* Warten bis alle Stationen bereit stehen *)
		200:	xTmp:=	(TStation_Work_St1.TControl.xDone OR TStation_Work_St1.TControl.xError);
			IF xTmp THEN
				xTmp:=	NOT(TStation_Work_St1.TControl.xError);
				IF xTmp THEN
					iStepFunction:=300;
				ELSE
					xStationErrorActive:=TRUE;
					iStepFunction:=999;
				END_IF;
			END_IF;
		(* Aktivieren der Prozessschicht *)
		300:	TProcess.T_Ctrle.xEnable:=TRUE;
			iStepFunction:=400;
		400:	IF TProcess.T_Ctrle.xRdy AND TProcess.T_Ctrle.xDone THEN
					iStepFunction:=600;
				END_IF;
		(* Lesen aller Profile *)
		600:	T_VisuQVis.T_CtrleAction.xExecute:=TRUE;
			T_VisuQVis.T_CtrleAction.iFunction:=1002;
			(* next step *)
			iStepFunction:=700;
		700:	IF NOT(T_VisuQVis.T_CtrleAction.xExecute) AND T_VisuQVis.T_CtrleAction.xDone THEN iStepFunction:=984; END_IF;
			IF NOT(T_VisuQVis.T_CtrleAction.xExecute) AND T_VisuQVis.T_CtrleAction.xErr THEN iStepFunction:=999; END_IF
			IF NOT(T_VisuQVis.T_CtrleAction.xExecute) AND (T_VisuQVis.T_CtrleAction.xDone OR T_VisuQVis.T_CtrleAction.xErr) THEN
				T_VisuQVis.T_PlcParam.dwSetNewPage:=16#A;	(* Main Page wird aufgerufen *)
				T_VisuQVis.T_CtrleVisu.iFunction:=1;
				T_VisuQVis.T_CtrleVisu.xExecute:=TRUE;
				gxAxisPositionSettled:=TRUE;	(* Achsen ref State der BIOS Parameter kann nun nicht mehr verstellt werden. Die Maschine muss zuerst ausgeschaltet werden
											    und muss wieder eingeschaltet werden. Vor dem erstmaligen Booten muss die Änderung der BIOS Parameter vorgenommen werden *)
			END_IF;
		984:	tTimeOutFunction:=T#0s;	(* deactivate the time out *)
			(* Overlay Message Info *)
			xMachineActivated:=TRUE;
			xActiveInfoMsgIntern:=TRUE;
			iStepFunctionMsg:=1;
			iMsgNumber:=1;		(* Modul wurde aufgestartet! Bestätigen Sie die Meldung und das Modul steht dann Bereit! *)
			(* next step *)
			iStepFunction:=985;
		985:	IF NOT(xActiveInfoMsgIntern) OR (T_TwinSafeIn.IxKeySwitchProcObservationCh1 AND T_TwinSafeIn.IxKeySwitchProcObservationCh2) OR (T_TwinSafeIn.IxKeySwitchWorkStationCh1 AND T_TwinSafeIn.IxKeySwitchWorkStationCh2) THEN
				T_ExchgParam.T_SafetyCtrl.bStateMessageInfo:=0;
				T_ExchgParam.T_SafetyCtrl.xConfirmMsgInfo:=FALSE;
				(* next step *)
				iStepFunction:=986;
			END_IF;
			T_StartUp.T_State.xCompleted:=TRUE;
		986:	T_ExchgParam.T_SafetyCtrl.xOpenSecurityDoorMachine:=TRUE;
			iStepFunction:=987;
		987:	IF NOT(T_ExchgParam.T_SafetyCtrl.xOpenSecurityDoorMachine) THEN
				iStepFunction:=990;
			END_IF;
		(* End function *)
		990:	T_StartUp.T_State.xCompleted:=TRUE;
			T_StartUp.T_State.xBlockChangeMovementVisu:=FALSE;
			T_StartUp.T_Ctrle.xDone:=TRUE;
			T_StartUp.T_Ctrle.xErr:=FALSE;
			T_StartUp.T_Ctrle.udiErrorID:=16#0;
			xLoading:=FALSE;
			tTimeOutFunction:=T#0s;	(* deactivate the time out *)
		(* Error function, set output disable *)
		999:	xActiveBootingError:=TRUE;
			tTimeOutFunction:=T#0s;	(* deactivate the time out *)
			TStation_Work_St1.TControl.xEnable:=FALSE;
			T_ExchgParam.T_Visu.iLoadingStartPage:=1;
			(* next step *)
			iStepFunction:=9994;
		9994:(* Overlay Message Error *)
			xActiveErrorMsgIntern:=TRUE;
			iStepFunctionMsg:=1;
			iMsgNumber:=49;		(* Während des Aufstarten der Maschine ist ein Fehler/Error aufgetreten! Bestätigen Sie die Meldung und Überprüfen Sie den entsprechenden Fehler/Error *)
			(* next step *)
			iStepFunction:=9995;
			T_TwinSafeCtrleOUT.xTwinSAFE_Run_1:=FALSE;	(* Stop TwinSafe Groupe 1 *)
		9995:IF NOT(xActiveErrorMsgIntern) THEN
				xStationErrorActive:=FALSE;
				(* next step *)
				iStepFunction:=9996;
			END_IF;
		9996:T_ExchgParam.T_SafetyCtrl.xOpenSecurityDoorMachine:=TRUE;
			iStepFunction:=9997;
		9997:IF NOT(T_ExchgParam.T_SafetyCtrl.xOpenSecurityDoorMachine) THEN
				iStepFunction:=9998;
			END_IF;
		9998:xLoading:=FALSE;
			xStartBooting:=TRUE;
			tTimeOutFunction:=T#0s;	(* deactivate the time out *)
			(* next step *)
			iStepFunction:=1;
		END_CASE
	END_IF
END_ACTION
ACTION StartUpFunction_MessageActivate:
xForceCloseMessage:=((T_TwinSafeIn.IxKeySwitchProcObservationCh1 AND T_TwinSafeIn.IxKeySwitchProcObservationCh2) OR (T_TwinSafeIn.IxKeySwitchWorkStationCh1 AND T_TwinSafeIn.IxKeySwitchWorkStationCh2)) AND T_StartUp.T_State.xCompleted;
(* Automode Process Page muss aufgerufen werden, falls der Automat Aktiv ist und man nicht auf dieser Seite steht *)
IF xActiveInfoMsg OR xActiveErrorMsg OR xActiveWarningMsg THEN
	xTmp:=	T_VisuQVis.T_CtrleVisu.xDone
			AND NOT(T_VisuQVis.T_CtrleVisu.xExecute)
			AND NOT(T_VisuQVis.T_CtrleVisu.xErr)
			AND (gT_PageNumber.iAutoMode_Process <> T_VisuQVis.T_PlcParam.dwActualPage)
			AND (gT_PageNumber.iAutoMode_ProcessValue1 <> T_VisuQVis.T_PlcParam.dwActualPage)
			AND (gT_PageNumber.iAutoMode_ProcessValue2 <> T_VisuQVis.T_PlcParam.dwActualPage)
			AND (gT_PageNumber.iAutoMode_PartQuality <> T_VisuQVis.T_PlcParam.dwActualPage)
			AND (TProcess.T_Ctrle.iFunctNr = 2)
			AND NOT(xForceCloseMessage) AND
			T_StartUp.T_State.xCompleted;
	IF xTmp THEN
		T_VisuQVis.T_CtrleVisu.iFunction:=1;
		T_VisuQVis.T_PlcParam.dwSetNewPage:=gT_PageNumber.iAutoMode_Process;
		T_VisuQVis.T_CtrleVisu.xExecute:=TRUE;
	END_IF;
END_IF;
(* Maschine Referenzierung Page muss aufgerufen werden, falls der Maschinen Referenzierung Aktiv ist und man nicht auf dieser Seite steht *)
IF xActiveInfoMsg OR xActiveErrorMsg OR xActiveWarningMsg THEN
	xTmp:=	T_VisuQVis.T_CtrleVisu.xDone
			AND NOT(T_VisuQVis.T_CtrleVisu.xExecute)
			AND NOT(T_VisuQVis.T_CtrleVisu.xErr)
			AND (gT_PageNumber.iAutoMode_Referencing <> T_VisuQVis.T_PlcParam.dwActualPage)
			AND (TProcess.T_Ctrle.iFunctNr = 1)
			AND NOT(xForceCloseMessage) AND
			T_StartUp.T_State.xCompleted;
	IF xTmp THEN
		T_VisuQVis.T_CtrleVisu.iFunction:=1;
		T_VisuQVis.T_PlcParam.dwSetNewPage:=gT_PageNumber.iAutoMode_Referencing;
		T_VisuQVis.T_CtrleVisu.xExecute:=TRUE;
	END_IF;
END_IF;

(* Acitvate Info Message Overlay *)
	IF xActiveInfoMsg OR xActiveInfoMsgIntern THEN
		CASE iStepFunctionMsg OF
		(* Check *)
		1:	T_StartUp.T_State.xBlockChangeMovementVisu:=TRUE;	(* Lock the navigation of the visu *)
			(* Overlay Message Error *)
			T_ExchgParam.T_SafetyCtrl.bStateMessageError:=0;
			T_ExchgParam.T_SafetyCtrl.bStateMessageInfo:=1;
			T_ExchgParam.T_SafetyCtrl.bStateMessageWarning:=0;
			T_ExchgParam.T_SafetyCtrl.iMsgInfoLine1:=iMsgNumber;
			T_ExchgParam.T_SafetyCtrl.iMsgInfoLine2:=iMsgNumber;
			T_ExchgParam.T_SafetyCtrl.iMsgInfoLine3:=iMsgNumber;
			T_ExchgParam.T_SafetyCtrl.iMsgInfoLine4:=iMsgNumber;
			T_ExchgParam.T_SafetyCtrl.xConfirmMsgInfo:=FALSE;
			(* next step *)
			iStepFunctionMsg:=iStepFunctionMsg + 1;
		2:	IF T_ExchgParam.T_SafetyCtrl.xConfirmMsgInfo OR xForceCloseMessage THEN
				xForceCloseMessage:=FALSE;
				T_StartUp.T_State.xBlockChangeMovementVisu:=FALSE;	(* Unlock the navigation of the visu *)
				T_ExchgParam.T_SafetyCtrl.bStateMessageInfo:=0;
				T_ExchgParam.T_SafetyCtrl.xConfirmMsgInfo:=FALSE;
				IF xActiveInfoMsg THEN
					T_StartUp.T_Ctrle.xDone:=TRUE;
					T_StartUp.T_Ctrle.xErr:=FALSE;
					T_StartUp.T_Ctrle.udiErrorID:=16#0;
				END_IF;
				xActiveInfoMsg:=FALSE;
				xActiveInfoMsgIntern:=FALSE;
				(* next step *)
				iStepFunctionMsg:=1;
				IF T_StartUp.T_Ctrle.xUnlockSecurityDoor THEN
					T_StartUp.T_Ctrle.xUnlockSecurityDoor:=FALSE;
					T_ExchgParam.T_SafetyCtrl.xOpenSecurityDoorMachine:=TRUE;
				END_IF;
			END_IF;
		END_CASE;
	END_IF;
	T_ExchgParam.T_SafetyCtrl.iMsgInfo_ColourState:=0;	(* Info Meldung mit grünem Hintergrund *)

(* Activate Error Message Overlay *)
	IF xActiveErrorMsg OR xActiveErrorMsgIntern THEN
		CASE iStepFunctionMsg OF
		(* Check *)
		1:	T_StartUp.T_State.xBlockChangeMovementVisu:=TRUE;	(* Lock the navigation of the visu *)
			(* Overlay Message Error *)
			T_ExchgParam.T_SafetyCtrl.bStateMessageError:=1;
			T_ExchgParam.T_SafetyCtrl.bStateMessageInfo:=0;
			T_ExchgParam.T_SafetyCtrl.bStateMessageWarning:=0;
			T_ExchgParam.T_SafetyCtrl.iMsgErrorLine1:=iMsgNumber;
			T_ExchgParam.T_SafetyCtrl.iMsgErrorLine2:=iMsgNumber;
			T_ExchgParam.T_SafetyCtrl.iMsgErrorLine3:=iMsgNumber;
			T_ExchgParam.T_SafetyCtrl.iMsgErrorLine4:=iMsgNumber;
			T_ExchgParam.T_SafetyCtrl.xConfirmMsgError:=FALSE;
			(* next step *)
			iStepFunctionMsg:=iStepFunctionMsg + 1;
		2:	IF T_ExchgParam.T_SafetyCtrl.xConfirmMsgError OR xForceCloseMessage THEN
				xForceCloseMessage:=FALSE;
				T_StartUp.T_State.xBlockChangeMovementVisu:=FALSE;	(* Unlock the navigation of the visu *)
				T_ExchgParam.T_SafetyCtrl.bStateMessageError:=0;
				T_ExchgParam.T_SafetyCtrl.xConfirmMsgError:=FALSE;
				IF xActiveErrorMsg THEN
					T_StartUp.T_Ctrle.xDone:=TRUE;
					T_StartUp.T_Ctrle.xErr:=FALSE;
					T_StartUp.T_Ctrle.udiErrorID:=16#0;
				END_IF;
				xActiveErrorMsg:=FALSE;
				xActiveErrorMsgIntern:=FALSE;
				(* next step *)
				iStepFunctionMsg:=1;
				IF T_StartUp.T_Ctrle.xUnlockSecurityDoor THEN
					T_StartUp.T_Ctrle.xUnlockSecurityDoor:=FALSE;
					T_ExchgParam.T_SafetyCtrl.xOpenSecurityDoorMachine:=TRUE;
				END_IF;
			END_IF;
		END_CASE;
	END_IF;

(* Activate Warning Message Overlay *)
	IF xActiveWarningMsg OR xActiveWarningMsgIntern THEN
		CASE iStepFunctionMsg OF
		(* Check *)
		1:	T_StartUp.T_State.xBlockChangeMovementVisu:=TRUE;	(* Lock the navigation of the visu *)
			(* Overlay Message Error *)
			T_ExchgParam.T_SafetyCtrl.bStateMessageError:=0;
			T_ExchgParam.T_SafetyCtrl.bStateMessageInfo:=0;
			T_ExchgParam.T_SafetyCtrl.bStateMessageWarning:=1;
			T_ExchgParam.T_SafetyCtrl.iMsgWarningLine1:=iMsgNumber;
			T_ExchgParam.T_SafetyCtrl.iMsgWarningLine2:=iMsgNumber;
			T_ExchgParam.T_SafetyCtrl.iMsgWarningLine3:=iMsgNumber;
			T_ExchgParam.T_SafetyCtrl.iMsgWarningLine4:=iMsgNumber;
			T_ExchgParam.T_SafetyCtrl.xConfirmMsgWarning:=FALSE;
			(* next step *)
			iStepFunctionMsg:=iStepFunctionMsg + 1;
		2:	IF T_ExchgParam.T_SafetyCtrl.xConfirmMsgWarning OR xForceCloseMessage THEN
				xForceCloseMessage:=FALSE;
				T_StartUp.T_State.xBlockChangeMovementVisu:=FALSE;	(* Unlock the navigation of the visu *)
				T_ExchgParam.T_SafetyCtrl.bStateMessageWarning:=0;
				T_ExchgParam.T_SafetyCtrl.xConfirmMsgWarning:=FALSE;
				IF xActiveWarningMsg THEN
					T_StartUp.T_Ctrle.xDone:=TRUE;
					T_StartUp.T_Ctrle.xErr:=FALSE;
					T_StartUp.T_Ctrle.udiErrorID:=16#0;
				END_IF;
				xActiveWarningMsg:=FALSE;
				xActiveWarningMsgIntern:=FALSE;
				(* next step *)
				iStepFunctionMsg:=1;
				IF T_StartUp.T_Ctrle.xUnlockSecurityDoor THEN
					T_StartUp.T_Ctrle.xUnlockSecurityDoor:=FALSE;
					T_ExchgParam.T_SafetyCtrl.xOpenSecurityDoorMachine:=TRUE;
				END_IF;
			END_IF;
		END_CASE;
	END_IF;

(* Löschen Aller Meldungen *)
	IF T_StartUp.T_Ctrle.xDeleteAllMessageOverlay AND (T_StartUp.T_State.xCompleted OR NOT(T_VisuQVis.T_CtrleVisu.xActive)) THEN
		T_StartUp.T_Ctrle.xDeleteAllMessageOverlay:=FALSE;
		xActiveInfoMsg:=xActiveInfoMsgIntern:=FALSE;
		xActiveErrorMsg:=xActiveErrorMsgIntern:=FALSE;
		xActiveWarningMsg:=xActiveWarningMsgIntern:=FALSE;
		T_ExchgParam.T_SafetyCtrl.bStateMessageError:=0;
		T_ExchgParam.T_SafetyCtrl.bStateMessageInfo:=0;
		T_ExchgParam.T_SafetyCtrl.bStateMessageWarning:=0;
		T_ExchgParam.T_SafetyCtrl.bStateMessageRequest:=0;
		T_ExchgParam.T_SafetyCtrl.bStateMessagePreWarning:=0;
		T_ExchgParam.T_SafetyCtrl.xConfirmMsgInfo:=FALSE;
		T_ExchgParam.T_SafetyCtrl.xConfirmMsgError:=FALSE;
		T_ExchgParam.T_SafetyCtrl.xConfirmMsgWarning:=FALSE;
		T_ExchgParam.T_SafetyCtrl.xConfirmMsgPreWarning:=FALSE;
		T_ExchgParam.T_SafetyCtrl.xConfirmMsgRequest:=FALSE;
		T_ExchgParam.T_SafetyCtrl.xConfirmMsgPartNumber:=FALSE;
		T_StartUp.T_State.xBlockChangeMovementVisu:=FALSE;
	ELSE
		T_StartUp.T_Ctrle.xDeleteAllMessageOverlay:=FALSE;
	END_IF;
END_ACTION
ACTION StartUpFunction_ReadHW:
(* Function ReadHardware with NovRAM Parameter *)
	IF xReadHardware THEN
		CASE iStepFunction OF
		(* Start station, reset FB *)
		1:	T_HDD.T_Ctrle.xReset:=TRUE;
			T_NovRAM.T_Ctrle.xReset:=TRUE;
			T_Profile.T_Ctrle.xReset:=TRUE;
			T_Password.T_Ctrle.xReset:=TRUE;
			T_ProcessData_St1.T_Ctrle.xReset:=TRUE;
			xNovRamParameterReaded:=FALSE;
			(* next step *)
			iStepFunction:=10;
			xNovRamError:=FALSE;
		(* waiting reset confirmation *)
		10:	xTmp:=	T_HDD.T_Ctrle.xDone
					AND T_NovRAM.T_Ctrle.xDone;
			IF xTmp THEN  iStepFunction:=20; END_IF
		(* Keine DeviceId mehr *)
		20:	(* next step *)
			iStepFunction:=30;
		(* waiting ID confirmation, Start BoxID *)
		30:	iStepFunction:=40;
		(* Keine BoxId mehr *)
		40:	iStepFunction:=50;
		50:	IF NOT(gxHardwareOFF) THEN
				T_NovRAM.T_Ctrle.iFunction:=1;
				T_NovRam.T_Ctrle.xBlockReadFirstTime:=FALSE;
				T_NovRAM.T_Ctrle.xExecute:=TRUE;
				T_NovRAM.T_Ctrle.tTimeOut:=T#5s;		(* IGS *) (* ansonsten erscheint Timeout NovRAM beim Booten *)
			END_IF;
			iStepFunction:=60;
		60:	IF NOT(T_NovRAM.T_Ctrle.xExecute) AND T_NovRAM.T_Ctrle.xDone THEN
				T_VisuQVis.T_CtrleVisu.xReset:=TRUE;
				iStepFunction:=70;
			END_IF;
			IF NOT(T_NovRAM.T_Ctrle.xExecute) AND T_NovRAM.T_Ctrle.xErr THEN
				xNovRamError:=TRUE;
				T_VisuQVis.T_CtrleVisu.xReset:=TRUE;
				T_NovRAM.T_Ctrle.xReset:=TRUE;
				iStepFunction:=99;
			END_IF;
		(* end function or time out *)
		70:	IF T_VisuQVis.T_CtrleVisu.xDone THEN
				T_StartUp.T_Ctrle.xDone:=TRUE;
				T_StartUp.T_Ctrle.xErr:=FALSE;
				T_StartUp.T_Ctrle.udiErrorID:=0;
				xReadHardware:=FALSE;
				tTimeOutFunction:=T#0s;
				(* Start Boot *)
				T_StartUp.T_Ctrle.xExecute:=TRUE;
				T_StartUp.T_Ctrle.iFunction:=5;
				xNovRamParameterReaded:=TRUE;
			END_IF;
		END_CASE;
	END_IF;
	T_ExchgParam.T_Config.xNoTouchScreenBtPanel:=NOT(gxHardwareOFF);;
END_ACTION

